LIN {X 0,Y 420.716,Z 380.039,A -85,B 0,C 180,E1 -10196.541,E2 -10196.541} C_VEL
LIN {X 0,Y 418.309,Z 369.381,A -85,B 0,C 180,E1 -10198.981,E2 -10198.981} C_VEL
LIN {X 0,Y 418.248,Z 369.386,A -85,B 0,C 180,E1 -10202.527,E2 -10202.527} C_VEL
LIN {X 0,Y 418.258,Z 369.383,A -85,B 0,C 180,E1 -10204.84,E2 -10204.84} C_VEL
LIN {X 0,Y 418.265,Z 369.379,A -85,B 0,C 180,E1 -10208.439,E2 -10208.439} C_VEL
LIN {X 0,Y 418.262,Z 369.382,A -85,B 0,C 180,E1 -10210.942,E2 -10210.942} C_VEL
LIN {X 0,Y 418.206,Z 369.391,A -85,B 0,C 180,E1 -10213.729,E2 -10213.729} C_VEL
LIN {X 0,Y 418.279,Z 369.382,A -85,B 0,C 180,E1 -10216.458,E2 -10216.458} C_VEL
LIN {X 0,Y 418.262,Z 369.383,A -85,B 0,C 180,E1 -10219.122,E2 -10219.122} C_VEL
LIN {X 0,Y 418.233,Z 369.387,A -85,B 0,C 180,E1 -10222.164,E2 -10222.164} C_VEL
LIN {X 0,Y 418.26,Z 369.385,A -85,B 0,C 180,E1 -10225.419,E2 -10225.419} C_VEL
LIN {X 0,Y 418.21,Z 369.387,A -85,B 0,C 180,E1 -10228.604,E2 -10228.604} C_VEL
LIN {X 0,Y 418.288,Z 369.381,A -85,B 0,C 180,E1 -10231.937,E2 -10231.937} C_VEL
LIN {X 0,Y 418.282,Z 369.378,A -85,B 0,C 180,E1 -10235.162,E2 -10235.162} C_VEL
LIN {X 0,Y 418.226,Z 369.382,A -85,B 0,C 180,E1 -10238.303,E2 -10238.303} C_VEL
LIN {X 0,Y 418.276,Z 369.385,A -85,B 0,C 180,E1 -10241.383,E2 -10241.383} C_VEL
LIN {X 0,Y 418.303,Z 369.376,A -85,B 0,C 180,E1 -10244.406,E2 -10244.406} C_VEL
LIN {X 0,Y 418.347,Z 369.369,A -85,B 0,C 180,E1 -10247.385,E2 -10247.385} C_VEL
LIN {X 0,Y 418.334,Z 369.373,A -85,B 0,C 180,E1 -10250.329,E2 -10250.329} C_VEL
LIN {X 0,Y 418.484,Z 369.351,A -85,B 0,C 180,E1 -10253.249,E2 -10253.249} C_VEL
LIN {X 0,Y 418.334,Z 369.377,A -85,B 0,C 180,E1 -10255.182,E2 -10255.182} C_VEL
LIN {X 0,Y 418.536,Z 369.344,A -85,B 0,C 180,E1 -10258.076,E2 -10258.076} C_VEL
LIN {X 0,Y 418.665,Z 369.332,A -85,B 0,C 180,E1 -10260,E2 -10260} C_VEL
LIN {X 0,Y 418.504,Z 369.347,A -85,B 0,C 180,E1 -10262.888,E2 -10262.888} C_VEL
LIN {X 0,Y 418.486,Z 369.354,A -85,B 0,C 180,E1 -10266.751,E2 -10266.751} C_VEL
LIN {X 0,Y 418.334,Z 369.375,A -85,B 0,C 180,E1 -10269.672,E2 -10269.672} C_VEL
LIN {X 0,Y 418.339,Z 369.371,A -85,B 0,C 180,E1 -10273.002,E2 -10273.002} C_VEL
LIN {X 0,Y 418.305,Z 369.373,A -85,B 0,C 180,E1 -10276.736,E2 -10276.736} C_VEL
LIN {X 0,Y 418.296,Z 369.374,A -85,B 0,C 180,E1 -10279.803,E2 -10279.803} C_VEL
LIN {X 0,Y 418.236,Z 369.389,A -85,B 0,C 180,E1 -10282.737,E2 -10282.737} C_VEL
LIN {X 0,Y 418.265,Z 369.382,A -85,B 0,C 180,E1 -10285.905,E2 -10285.905} C_VEL
LIN {X 0,Y 418.259,Z 369.385,A -85,B 0,C 180,E1 -10289.163,E2 -10289.163} C_VEL
LIN {X 0,Y 418.253,Z 369.384,A -85,B 0,C 180,E1 -10292.845,E2 -10292.845} C_VEL
LIN {X 0,Y 418.245,Z 369.385,A -85,B 0,C 180,E1 -10296.24,E2 -10296.24} C_VEL
LIN {X 0,Y 418.262,Z 369.381,A -85,B 0,C 180,E1 -10299.681,E2 -10299.681} C_VEL
LIN {X 0,Y 418.283,Z 369.377,A -85,B 0,C 180,E1 -10302.331,E2 -10302.331} C_VEL
LIN {X 0,Y 418.253,Z 369.383,A -85,B 0,C 180,E1 -10305.112,E2 -10305.112} C_VEL
LIN {X 0,Y 418.241,Z 369.385,A -85,B 0,C 180,E1 -10307.768,E2 -10307.768} C_VEL
LIN {X 0,Y 418.309,Z 369.47,A -85,B 0,C 180,E1 -10311.605,E2 -10311.605} C_VEL
LIN {X 0,Y 420.342,Z 380.03,A -85,B 0,C 180,E1 -10314.486,E2 -10314.486} C_VEL
LIN {X 0,Y 420.452,Z 381.221,A -85,B 0,C 180,E1 -10314.727,E2 -10314.727} C_VEL
LIN {X 0,Y 424.73,Z 398.892,A -85,B 0,C 180,E1 -10315.282,E2 -10315.282} C_VEL
LIN {X 0,Y 423.561,Z 487.472,A -85,B 0,C 180,E1 -10316.837,E2 -10316.837} C_VEL
LIN {X 0,Y 423.153,Z 500.671,A -85,B 0,C 180,E1 -10317.261,E2 -10317.261} C_VEL
LIN {X 0,Y 422.674,Z 513.047,A -85,B 0,C 180,E1 -10317.855,E2 -10317.855} C_VEL
LIN {X 0,Y 422.08,Z 523.932,A -85,B 0,C 180,E1 -10318.551,E2 -10318.551} C_VEL
LIN {X 0,Y 421.366,Z 534.615,A -85,B 0,C 180,E1 -10319.423,E2 -10319.423} C_VEL
LIN {X 0,Y 420.629,Z 544.481,A -85,B 0,C 180,E1 -10320.424,E2 -10320.424} C_VEL
LIN {X 0,Y 419.909,Z 553.272,A -85,B 0,C 180,E1 -10321.511,E2 -10321.511} C_VEL
LIN {X 0,Y 419.255,Z 561.69,A -85,B 0,C 180,E1 -10322.78,E2 -10322.78} C_VEL
LIN {X 0,Y 418.625,Z 568.972,A -85,B 0,C 180,E1 -10324.12,E2 -10324.12} C_VEL
LIN {X 0,Y 418.115,Z 575.775,A -85,B 0,C 180,E1 -10325.682,E2 -10325.682} C_VEL
LIN {X 0,Y 417.7,Z 581.039,A -85,B 0,C 180,E1 -10327.234,E2 -10327.234} C_VEL
LIN {X 0,Y 417.393,Z 585.027,A -85,B 0,C 180,E1 -10328.777,E2 -10328.777} C_VEL
LIN {X 0,Y 417.135,Z 588.367,A -85,B 0,C 180,E1 -10330.65,E2 -10330.65} C_VEL
LIN {X 0,Y 416.988,Z 590.049,A -85,B 0,C 180,E1 -10332.34,E2 -10332.34} C_VEL
LIN {X 0,Y 416.977,Z 590.52,A -85,B 0,C 180,E1 -10333.889,E2 -10333.889} C_VEL
LIN {X 0,Y 416.966,Z 590.033,A -85,B 0,C 180,E1 -10335.356,E2 -10335.356} C_VEL
LIN {X 0,Y 417.019,Z 589.173,A -85,B 0,C 180,E1 -10336.353,E2 -10336.353} C_VEL
LIN {X 0,Y 417.154,Z 587.301,A -85,B 0,C 180,E1 -10337.732,E2 -10337.732} C_VEL
LIN {X 0,Y 417.354,Z 584.039,A -85,B 0,C 180,E1 -10339.325,E2 -10339.325} C_VEL
LIN {X 0,Y 417.548,Z 579.915,A -85,B 0,C 180,E1 -10340.799,E2 -10340.799} C_VEL
LIN {X 0,Y 417.895,Z 574.601,A -85,B 0,C 180,E1 -10342.268,E2 -10342.268} C_VEL
LIN {X 0,Y 418.033,Z 572.633,A -85,B 0,C 180,E1 -10342.74,E2 -10342.74} C_VEL
LIN {X 0,Y 417.574,Z 569.57,A -85,B 0,C 180,E1 -10343.426,E2 -10343.426} C_VEL
LIN {X 0,Y 415.078,Z 564.217,A -85,B 0,C 180,E1 -10344.53,E2 -10344.53} C_VEL
LIN {X 0,Y 412.642,Z 558.354,A -85,B 0,C 180,E1 -10345.586,E2 -10345.586} C_VEL
LIN {X 0,Y 412.275,Z 554.353,A -85,B 0,C 180,E1 -10346.187,E2 -10346.187} C_VEL
LIN {X 0,Y 412.984,Z 544.392,A -85,B 0,C 180,E1 -10347.44,E2 -10347.44} C_VEL
LIN {X 0,Y 413.712,Z 533.485,A -85,B 0,C 180,E1 -10348.54,E2 -10348.54} C_VEL
LIN {X 0,Y 414.406,Z 522.256,A -85,B 0,C 180,E1 -10349.429,E2 -10349.429} C_VEL
LIN {X 0,Y 415,Z 509.859,A -85,B 0,C 180,E1 -10350.186,E2 -10350.186} C_VEL
LIN {X 0,Y 415.435,Z 497.781,A -85,B 0,C 180,E1 -10350.725,E2 -10350.725} C_VEL
LIN {X 0,Y 415.687,Z 484.799,A -85,B 0,C 180,E1 -10351.1,E2 -10351.1} C_VEL
LIN {X 0,Y 416.747,Z 399.82,A -85,B 0,C 180,E1 -10352.579,E2 -10352.579} C_VEL
LIN {X 0,Y 412.903,Z 380.764,A -85,B 0,C 180,E1 -10353.079,E2 -10353.079} C_VEL
LIN {X 0,Y 412.963,Z 379.392,A -85,B 0,C 180,E1 -10353.415,E2 -10353.415} C_VEL
LIN {X 0,Y 411.478,Z 370.232,A -85,B 0,C 180,E1 -10355.82,E2 -10355.82} C_VEL
LIN {X 0,Y 411.324,Z 370.25,A -85,B 0,C 180,E1 -10358.846,E2 -10358.846} C_VEL
LIN {X 0,Y 411.29,Z 370.251,A -85,B 0,C 180,E1 -10361.832,E2 -10361.832} C_VEL
LIN {X 0,Y 411.266,Z 370.254,A -85,B 0,C 180,E1 -10364.852,E2 -10364.852} C_VEL
LIN {X 0,Y 411.257,Z 370.254,A -85,B 0,C 180,E1 -10367.914,E2 -10367.914} C_VEL
LIN {X 0,Y 411.2,Z 370.264,A -85,B 0,C 180,E1 -10371.033,E2 -10371.033} C_VEL
LIN {X 0,Y 411.23,Z 370.256,A -85,B 0,C 180,E1 -10374.215,E2 -10374.215} C_VEL
LIN {X 0,Y 411.261,Z 370.257,A -85,B 0,C 180,E1 -10377.477,E2 -10377.477} C_VEL
LIN {X 0,Y 411.2,Z 370.263,A -85,B 0,C 180,E1 -10380.846,E2 -10380.846} C_VEL
LIN {X 0,Y 411.207,Z 370.259,A -85,B 0,C 180,E1 -10384.332,E2 -10384.332} C_VEL
LIN {X 0,Y 411.202,Z 370.26,A -85,B 0,C 180,E1 -10387.972,E2 -10387.972} C_VEL
LIN {X 0,Y 411.183,Z 370.263,A -85,B 0,C 180,E1 -10390.503,E2 -10390.503} C_VEL
LIN {X 0,Y 411.172,Z 370.27,A -85,B 0,C 180,E1 -10393.133,E2 -10393.133} C_VEL
LIN {X 0,Y 411.171,Z 370.264,A -85,B 0,C 180,E1 -10395.879,E2 -10395.879} C_VEL
LIN {X 0,Y 411.163,Z 370.269,A -85,B 0,C 180,E1 -10398.77,E2 -10398.77} C_VEL
LIN {X 0,Y 411.208,Z 370.259,A -85,B 0,C 180,E1 -10401.829,E2 -10401.829} C_VEL
LIN {X 0,Y 411.207,Z 370.264,A -85,B 0,C 180,E1 -10405.12,E2 -10405.12} C_VEL
LIN {X 0,Y 411.161,Z 370.265,A -85,B 0,C 180,E1 -10408.002,E2 -10408.002} C_VEL
LIN {X 0,Y 411.212,Z 370.26,A -85,B 0,C 180,E1 -10411.409,E2 -10411.409} C_VEL
LIN {X 0,Y 411.232,Z 370.256,A -85,B 0,C 180,E1 -10413.618,E2 -10413.618} C_VEL
LIN {X 0,Y 411.197,Z 370.267,A -85,B 0,C 180,E1 -10416.852,E2 -10416.852} C_VEL
LIN {X 0,Y 411.208,Z 370.26,A -85,B 0,C 180,E1 -10420.05,E2 -10420.05} C_VEL
LIN {X 0,Y 411.256,Z 370.256,A -85,B 0,C 180,E1 -10423.13,E2 -10423.13} C_VEL
LIN {X 0,Y 411.298,Z 370.252,A -85,B 0,C 180,E1 -10426.895,E2 -10426.895} C_VEL
LIN {X 0,Y 411.286,Z 370.251,A -85,B 0,C 180,E1 -10430.161,E2 -10430.161} C_VEL
LIN {X 0,Y 411.448,Z 370.231,A -85,B 0,C 180,E1 -10433.133,E2 -10433.133} C_VEL
LIN {X 0,Y 411.306,Z 370.249,A -85,B 0,C 180,E1 -10435.099,E2 -10435.099} C_VEL
LIN {X 0,Y 411.506,Z 370.224,A -85,B 0,C 180,E1 -10438.042,E2 -10438.042} C_VEL
LIN {X 0,Y 411.633,Z 370.208,A -85,B 0,C 180,E1 -10440,E2 -10440} C_VEL
LIN {X 0,Y 411.458,Z 370.23,A -85,B 0,C 180,E1 -10442.937,E2 -10442.937} C_VEL
LIN {X 0,Y 411.447,Z 370.232,A -85,B 0,C 180,E1 -10446.867,E2 -10446.867} C_VEL
LIN {X 0,Y 411.285,Z 370.251,A -85,B 0,C 180,E1 -10449.839,E2 -10449.839} C_VEL
LIN {X 0,Y 411.297,Z 370.248,A -85,B 0,C 180,E1 -10453.104,E2 -10453.104} C_VEL
LIN {X 0,Y 411.256,Z 370.255,A -85,B 0,C 180,E1 -10456.87,E2 -10456.87} C_VEL
LIN {X 0,Y 411.222,Z 370.261,A -85,B 0,C 180,E1 -10459.987,E2 -10459.987} C_VEL
LIN {X 0,Y 411.195,Z 370.261,A -85,B 0,C 180,E1 -10463.148,E2 -10463.148} C_VEL
LIN {X 0,Y 411.231,Z 370.262,A -85,B 0,C 180,E1 -10466.381,E2 -10466.381} C_VEL
LIN {X 0,Y 411.204,Z 370.262,A -85,B 0,C 180,E1 -10469.712,E2 -10469.712} C_VEL
LIN {X 0,Y 411.2,Z 370.26,A -85,B 0,C 180,E1 -10473.156,E2 -10473.156} C_VEL
LIN {X 0,Y 411.19,Z 370.264,A -85,B 0,C 180,E1 -10476.554,E2 -10476.554} C_VEL
LIN {X 0,Y 411.224,Z 370.26,A -85,B 0,C 180,E1 -10479.731,E2 -10479.731} C_VEL
LIN {X 0,Y 411.226,Z 370.257,A -85,B 0,C 180,E1 -10483.127,E2 -10483.127} C_VEL
LIN {X 0,Y 411.168,Z 370.27,A -85,B 0,C 180,E1 -10485.881,E2 -10485.881} C_VEL
LIN {X 0,Y 411.209,Z 370.261,A -85,B 0,C 180,E1 -10489.5,E2 -10489.5} C_VEL
LIN {X 0,Y 411.203,Z 370.266,A -85,B 0,C 180,E1 -10492.028,E2 -10492.028} C_VEL
LIN {X 0,Y 411.205,Z 370.264,A -85,B 0,C 180,E1 -10495.667,E2 -10495.667} C_VEL
LIN {X 0,Y 411.199,Z 370.261,A -85,B 0,C 180,E1 -10499.154,E2 -10499.154} C_VEL
LIN {X 0,Y 411.326,Z 370.37,A -85,B 0,C 180,E1 -10501.767,E2 -10501.767} C_VEL
LIN {X 0,Y 413.906,Z 383.596,A -85,B 0,C 180,E1 -10504.566,E2 -10504.566} C_VEL
LIN {X 0,Y 414.291,Z 387.926,A -85,B 0,C 180,E1 -10505.443,E2 -10505.443} C_VEL
LIN {X 0,Y 413.242,Z 404.064,A -85,B 0,C 180,E1 -10508.553,E2 -10508.553} C_VEL
LIN {X 0,Y 412.459,Z 416.368,A -85,B 0,C 180,E1 -10510.901,E2 -10510.901} C_VEL
LIN {X 0,Y 416.383,Z 444.904,A -85,B 0,C 180,E1 -10511.566,E2 -10511.566} C_VEL
LIN {X 0,Y 415.489,Z 524.864,A -85,B 0,C 180,E1 -10512.972,E2 -10512.972} C_VEL
LIN {X 0,Y 414.979,Z 538.176,A -85,B 0,C 180,E1 -10513.394,E2 -10513.394} C_VEL
LIN {X 0,Y 414.344,Z 550.959,A -85,B 0,C 180,E1 -10514.001,E2 -10514.001} C_VEL
LIN {X 0,Y 413.64,Z 562.314,A -85,B 0,C 180,E1 -10514.731,E2 -10514.731} C_VEL
LIN {X 0,Y 412.865,Z 574.043,A -85,B 0,C 180,E1 -10515.711,E2 -10515.711} C_VEL
LIN {X 0,Y 412.266,Z 583.918,A -85,B 0,C 180,E1 -10516.741,E2 -10516.741} C_VEL
LIN {X 0,Y 411.637,Z 593.223,A -85,B 0,C 180,E1 -10517.928,E2 -10517.928} C_VEL
LIN {X 0,Y 411.014,Z 601.161,A -85,B 0,C 180,E1 -10519.159,E2 -10519.159} C_VEL
LIN {X 0,Y 410.569,Z 608.912,A -85,B 0,C 180,E1 -10520.641,E2 -10520.641} C_VEL
LIN {X 0,Y 410.27,Z 615.134,A -85,B 0,C 180,E1 -10522.124,E2 -10522.124} C_VEL
LIN {X 0,Y 410.089,Z 620.393,A -85,B 0,C 180,E1 -10523.716,E2 -10523.716} C_VEL
LIN {X 0,Y 410.048,Z 623.859,A -85,B 0,C 180,E1 -10525.084,E2 -10525.084} C_VEL
LIN {X 0,Y 409.947,Z 625.807,A -85,B 0,C 180,E1 -10526.068,E2 -10526.068} C_VEL
LIN {X 0,Y 409.989,Z 627.336,A -85,B 0,C 180,E1 -10527.052,E2 -10527.052} C_VEL
LIN {X 0,Y 410.019,Z 628.405,A -85,B 0,C 180,E1 -10528.035,E2 -10528.035} C_VEL
LIN {X 0,Y 409.972,Z 629.35,A -85,B 0,C 180,E1 -10530,E2 -10530} C_VEL
LIN {X 0,Y 409.978,Z 629.236,A -85,B 0,C 180,E1 -10530.982,E2 -10530.982} C_VEL
LIN {X 0,Y 410.018,Z 628.688,A -85,B 0,C 180,E1 -10531.965,E2 -10531.965} C_VEL
LIN {X 0,Y 409.97,Z 627.738,A -85,B 0,C 180,E1 -10532.948,E2 -10532.948} C_VEL
LIN {X 0,Y 410.025,Z 624.641,A -85,B 0,C 180,E1 -10534.916,E2 -10534.916} C_VEL
LIN {X 0,Y 410.041,Z 621.58,A -85,B 0,C 180,E1 -10536.224,E2 -10536.224} C_VEL
LIN {X 0,Y 410.284,Z 616.556,A -85,B 0,C 180,E1 -10537.876,E2 -10537.876} C_VEL
LIN {X 0,Y 410.674,Z 609.634,A -85,B 0,C 180,E1 -10539.605,E2 -10539.605} C_VEL
LIN {X 0,Y 411.257,Z 602.158,A -85,B 0,C 180,E1 -10541.084,E2 -10541.084} C_VEL
LIN {X 0,Y 411.897,Z 594.555,A -85,B 0,C 180,E1 -10542.314,E2 -10542.314} C_VEL
LIN {X 0,Y 412.576,Z 585.369,A -85,B 0,C 180,E1 -10543.546,E2 -10543.546} C_VEL
LIN {X 0,Y 413.385,Z 575.315,A -85,B 0,C 180,E1 -10544.636,E2 -10544.636} C_VEL
LIN {X 0,Y 414.315,Z 563.918,A -85,B 0,C 180,E1 -10545.621,E2 -10545.621} C_VEL
LIN {X 0,Y 415.242,Z 551.273,A -85,B 0,C 180,E1 -10546.468,E2 -10546.468} C_VEL
LIN {X 0,Y 416.025,Z 538.172,A -85,B 0,C 180,E1 -10547.1,E2 -10547.1} C_VEL
LIN {X 0,Y 416.546,Z 525.252,A -85,B 0,C 180,E1 -10547.521,E2 -10547.521} C_VEL
LIN {X 0,Y 417.586,Z 444.003,A -85,B 0,C 180,E1 -10548.979,E2 -10548.979} C_VEL
LIN {X 0,Y 414.204,Z 422.378,A -85,B 0,C 180,E1 -10549.561,E2 -10549.561} C_VEL
LIN {X 0,Y 413.002,Z 415.847,A -85,B 0,C 180,E1 -10549.753,E2 -10549.753} C_VEL
LIN {X 0,Y 414.378,Z 397.592,A -85,B 0,C 180,E1 -10553.344,E2 -10553.344} C_VEL
LIN {X 0,Y 415.039,Z 389.085,A -85,B 0,C 180,E1 -10555.045,E2 -10555.045} C_VEL
LIN {X 0,Y 413.784,Z 381.321,A -85,B 0,C 180,E1 -10556.749,E2 -10556.749} C_VEL
LIN {X 0,Y 411.229,Z 370.261,A -85,B 0,C 180,E1 -10559.354,E2 -10559.354} C_VEL
LIN {X 0,Y 411.205,Z 370.26,A -85,B 0,C 180,E1 -10563.155,E2 -10563.155} C_VEL
LIN {X 0,Y 411.194,Z 370.267,A -85,B 0,C 180,E1 -10566.553,E2 -10566.553} C_VEL
LIN {X 0,Y 411.226,Z 370.26,A -85,B 0,C 180,E1 -10569.73,E2 -10569.73} C_VEL
LIN {X 0,Y 411.173,Z 370.263,A -85,B 0,C 180,E1 -10573.132,E2 -10573.132} C_VEL
LIN {X 0,Y 411.231,Z 370.261,A -85,B 0,C 180,E1 -10575.871,E2 -10575.871} C_VEL
LIN {X 0,Y 411.205,Z 370.262,A -85,B 0,C 180,E1 -10578.764,E2 -10578.764} C_VEL
LIN {X 0,Y 411.2,Z 370.264,A -85,B 0,C 180,E1 -10582.027,E2 -10582.027} C_VEL
LIN {X 0,Y 411.2,Z 370.264,A -85,B 0,C 180,E1 -10585.666,E2 -10585.666} C_VEL
LIN {X 0,Y 411.191,Z 370.263,A -85,B 0,C 180,E1 -10589.153,E2 -10589.153} C_VEL
LIN {X 0,Y 411.253,Z 370.254,A -85,B 0,C 180,E1 -10592.522,E2 -10592.522} C_VEL
LIN {X 0,Y 411.22,Z 370.264,A -85,B 0,C 180,E1 -10595.784,E2 -10595.784} C_VEL
LIN {X 0,Y 411.188,Z 370.258,A -85,B 0,C 180,E1 -10598.966,E2 -10598.966} C_VEL
LIN {X 0,Y 411.245,Z 370.251,A -85,B 0,C 180,E1 -10602.085,E2 -10602.085} C_VEL
LIN {X 0,Y 411.257,Z 370.257,A -85,B 0,C 180,E1 -10605.147,E2 -10605.147} C_VEL
LIN {X 0,Y 411.276,Z 370.249,A -85,B 0,C 180,E1 -10608.167,E2 -10608.167} C_VEL
LIN {X 0,Y 411.432,Z 370.225,A -85,B 0,C 180,E1 -10612.189,E2 -10612.189} C_VEL
LIN {X 0,Y 411.467,Z 370.228,A -85,B 0,C 180,E1 -10614.118,E2 -10614.118} C_VEL
LIN {X 0,Y 411.505,Z 370.22,A -85,B 0,C 180,E1 -10618.043,E2 -10618.043} C_VEL
LIN {X 0,Y 411.635,Z 370.208,A -85,B 0,C 180,E1 -10620,E2 -10620} C_VEL
LIN {X 0,Y 411.46,Z 370.224,A -85,B 0,C 180,E1 -10622.937,E2 -10622.937} C_VEL
LIN {X 0,Y 411.453,Z 370.23,A -85,B 0,C 180,E1 -10626.867,E2 -10626.867} C_VEL
LIN {X 0,Y 411.286,Z 370.251,A -85,B 0,C 180,E1 -10629.839,E2 -10629.839} C_VEL
LIN {X 0,Y 411.298,Z 370.249,A -85,B 0,C 180,E1 -10633.105,E2 -10633.105} C_VEL
LIN {X 0,Y 411.256,Z 370.252,A -85,B 0,C 180,E1 -10636.87,E2 -10636.87} C_VEL
LIN {X 0,Y 411.249,Z 370.251,A -85,B 0,C 180,E1 -10639.986,E2 -10639.986} C_VEL
LIN {X 0,Y 411.2,Z 370.262,A -85,B 0,C 180,E1 -10643.148,E2 -10643.148} C_VEL
LIN {X 0,Y 411.232,Z 370.259,A -85,B 0,C 180,E1 -10646.382,E2 -10646.382} C_VEL
LIN {X 0,Y 411.195,Z 370.261,A -85,B 0,C 180,E1 -10649.714,E2 -10649.714} C_VEL
LIN {X 0,Y 411.202,Z 370.257,A -85,B 0,C 180,E1 -10653.157,E2 -10653.157} C_VEL
LIN {X 0,Y 411.192,Z 370.266,A -85,B 0,C 180,E1 -10656.554,E2 -10656.554} C_VEL
LIN {X 0,Y 411.224,Z 370.258,A -85,B 0,C 180,E1 -10659.731,E2 -10659.731} C_VEL
LIN {X 0,Y 411.226,Z 370.262,A -85,B 0,C 180,E1 -10663.127,E2 -10663.127} C_VEL
LIN {X 0,Y 411.175,Z 370.266,A -85,B 0,C 180,E1 -10665.881,E2 -10665.881} C_VEL
LIN {X 0,Y 411.165,Z 370.271,A -85,B 0,C 180,E1 -10668.772,E2 -10668.772} C_VEL
LIN {X 0,Y 411.245,Z 370.355,A -85,B 0,C 180,E1 -10671.29,E2 -10671.29} C_VEL
LIN {X 0,Y 413.427,Z 381.383,A -85,B 0,C 180,E1 -10674.329,E2 -10674.329} C_VEL
LIN {X 0,Y 417.054,Z 395.122,A -85,B 0,C 180,E1 -10674.791,E2 -10674.791} C_VEL
LIN {X 0,Y 418.228,Z 400.694,A -85,B 0,C 180,E1 -10674.959,E2 -10674.959} C_VEL
LIN {X 0,Y 416.923,Z 487.236,A -85,B 0,C 180,E1 -10676.492,E2 -10676.492} C_VEL
LIN {X 0,Y 416.51,Z 500.636,A -85,B 0,C 180,E1 -10676.925,E2 -10676.925} C_VEL
LIN {X 0,Y 416.017,Z 512.437,A -85,B 0,C 180,E1 -10677.49,E2 -10677.49} C_VEL
LIN {X 0,Y 415.335,Z 524.449,A -85,B 0,C 180,E1 -10678.263,E2 -10678.263} C_VEL
LIN {X 0,Y 414.577,Z 535.101,A -85,B 0,C 180,E1 -10679.15,E2 -10679.15} C_VEL
LIN {X 0,Y 413.682,Z 546.359,A -85,B 0,C 180,E1 -10680.332,E2 -10680.332} C_VEL
LIN {X 0,Y 412.87,Z 555.591,A -85,B 0,C 180,E1 -10681.536,E2 -10681.536} C_VEL
LIN {X 0,Y 412.182,Z 563.863,A -85,B 0,C 180,E1 -10682.865,E2 -10682.865} C_VEL
LIN {X 0,Y 411.431,Z 571.792,A -85,B 0,C 180,E1 -10684.45,E2 -10684.45} C_VEL
LIN {X 0,Y 411.009,Z 577.104,A -85,B 0,C 180,E1 -10685.772,E2 -10685.772} C_VEL
LIN {X 0,Y 410.615,Z 581.904,A -85,B 0,C 180,E1 -10687.261,E2 -10687.261} C_VEL
LIN {X 0,Y 410.296,Z 585.943,A -85,B 0,C 180,E1 -10688.918,E2 -10688.918} C_VEL
LIN {X 0,Y 410.064,Z 588.629,A -85,B 0,C 180,E1 -10690.5,E2 -10690.5} C_VEL
LIN {X 0,Y 409.914,Z 590.203,A -85,B 0,C 180,E1 -10692.025,E2 -10692.025} C_VEL
LIN {X 0,Y 409.894,Z 590.853,A -85,B 0,C 180,E1 -10693.777,E2 -10693.777} C_VEL
LIN {X 0,Y 409.891,Z 590.487,A -85,B 0,C 180,E1 -10695.097,E2 -10695.097} C_VEL
LIN {X 0,Y 409.904,Z 589.756,A -85,B 0,C 180,E1 -10696.112,E2 -10696.112} C_VEL
LIN {X 0,Y 410.066,Z 587.775,A -85,B 0,C 180,E1 -10697.665,E2 -10697.665} C_VEL
LIN {X 0,Y 410.243,Z 584.921,A -85,B 0,C 180,E1 -10699.138,E2 -10699.138} C_VEL
LIN {X 0,Y 410.451,Z 580.973,A -85,B 0,C 180,E1 -10700.639,E2 -10700.639} C_VEL
LIN {X 0,Y 410.801,Z 575.871,A -85,B 0,C 180,E1 -10702.134,E2 -10702.134} C_VEL
LIN {X 0,Y 411.193,Z 569.457,A -85,B 0,C 180,E1 -10703.622,E2 -10703.622} C_VEL
LIN {X 0,Y 411.758,Z 561.444,A -85,B 0,C 180,E1 -10705.104,E2 -10705.104} C_VEL
LIN {X 0,Y 412.275,Z 554.353,A -85,B 0,C 180,E1 -10706.187,E2 -10706.187} C_VEL
LIN {X 0,Y 411.937,Z 550.209,A -85,B 0,C 180,E1 -10706.764,E2 -10706.764} C_VEL
LIN {X 0,Y 409.649,Z 543.204,A -85,B 0,C 180,E1 -10707.689,E2 -10707.689} C_VEL
LIN {X 0,Y 407.351,Z 535.723,A -85,B 0,C 180,E1 -10708.546,E2 -10708.546} C_VEL
LIN {X 0,Y 406.998,Z 530.789,A -85,B 0,C 180,E1 -10709.011,E2 -10709.011} C_VEL
LIN {X 0,Y 407.728,Z 519.319,A -85,B 0,C 180,E1 -10709.878,E2 -10709.878} C_VEL
LIN {X 0,Y 408.226,Z 506.943,A -85,B 0,C 180,E1 -10710.585,E2 -10710.585} C_VEL
LIN {X 0,Y 408.664,Z 493.988,A -85,B 0,C 180,E1 -10711.109,E2 -10711.109} C_VEL
LIN {X 0,Y 408.949,Z 481.779,A -85,B 0,C 180,E1 -10711.416,E2 -10711.416} C_VEL
LIN {X 0,Y 409.897,Z 400.575,A -85,B 0,C 180,E1 -10712.845,E2 -10712.845} C_VEL
LIN {X 0,Y 405.956,Z 381.024,A -85,B 0,C 180,E1 -10713.377,E2 -10713.377} C_VEL
LIN {X 0,Y 404.398,Z 371.113,A -85,B 0,C 180,E1 -10715.985,E2 -10715.985} C_VEL
LIN {X 0,Y 404.271,Z 371.129,A -85,B 0,C 180,E1 -10719.001,E2 -10719.001} C_VEL
LIN {X 0,Y 404.262,Z 371.125,A -85,B 0,C 180,E1 -10722.041,E2 -10722.041} C_VEL
LIN {X 0,Y 404.212,Z 371.135,A -85,B 0,C 180,E1 -10725.117,E2 -10725.117} C_VEL
LIN {X 0,Y 404.214,Z 371.13,A -85,B 0,C 180,E1 -10728.237,E2 -10728.237} C_VEL
LIN {X 0,Y 404.164,Z 371.142,A -85,B 0,C 180,E1 -10731.417,E2 -10731.417} C_VEL
LIN {X 0,Y 404.18,Z 371.136,A -85,B 0,C 180,E1 -10734.665,E2 -10734.665} C_VEL
LIN {X 0,Y 404.198,Z 371.133,A -85,B 0,C 180,E1 -10737.999,E2 -10737.999} C_VEL
LIN {X 0,Y 404.148,Z 371.141,A -85,B 0,C 180,E1 -10741.559,E2 -10741.559} C_VEL
LIN {X 0,Y 404.186,Z 371.139,A -85,B 0,C 180,E1 -10745.015,E2 -10745.015} C_VEL
LIN {X 0,Y 404.16,Z 371.14,A -85,B 0,C 180,E1 -10748.755,E2 -10748.755} C_VEL
LIN {X 0,Y 404.122,Z 371.143,A -85,B 0,C 180,E1 -10751.599,E2 -10751.599} C_VEL
LIN {X 0,Y 404.145,Z 371.141,A -85,B 0,C 180,E1 -10754.521,E2 -10754.521} C_VEL
LIN {X 0,Y 404.137,Z 371.143,A -85,B 0,C 180,E1 -10757.295,E2 -10757.295} C_VEL
LIN {X 0,Y 404.166,Z 371.136,A -85,B 0,C 180,E1 -10759.954,E2 -10759.954} C_VEL
LIN {X 0,Y 404.137,Z 371.145,A -85,B 0,C 180,E1 -10763.123,E2 -10763.123} C_VEL
LIN {X 0,Y 404.141,Z 371.14,A -85,B 0,C 180,E1 -10766.187,E2 -10766.187} C_VEL
LIN {X 0,Y 404.14,Z 371.14,A -85,B 0,C 180,E1 -10769.714,E2 -10769.714} C_VEL
LIN {X 0,Y 404.19,Z 371.137,A -85,B 0,C 180,E1 -10773.122,E2 -10773.122} C_VEL
LIN {X 0,Y 404.171,Z 371.137,A -85,B 0,C 180,E1 -10775.334,E2 -10775.334} C_VEL
LIN {X 0,Y 404.132,Z 371.145,A -85,B 0,C 180,E1 -10778.58,E2 -10778.58} C_VEL
LIN {X 0,Y 404.203,Z 371.132,A -85,B 0,C 180,E1 -10781.761,E2 -10781.761} C_VEL
LIN {X 0,Y 404.201,Z 371.137,A -85,B 0,C 180,E1 -10784.881,E2 -10784.881} C_VEL
LIN {X 0,Y 404.25,Z 371.126,A -85,B 0,C 180,E1 -10787.958,E2 -10787.958} C_VEL
LIN {X 0,Y 404.397,Z 371.109,A -85,B 0,C 180,E1 -10792.128,E2 -10792.128} C_VEL
LIN {X 0,Y 404.416,Z 371.106,A -85,B 0,C 180,E1 -10794.015,E2 -10794.015} C_VEL
LIN {X 0,Y 404.475,Z 371.099,A -85,B 0,C 180,E1 -10798.008,E2 -10798.008} C_VEL
LIN {X 0,Y 404.602,Z 371.084,A -85,B 0,C 180,E1 -10800,E2 -10800} C_VEL
LIN {X 0,Y 404.415,Z 371.107,A -85,B 0,C 180,E1 -10802.988,E2 -10802.988} C_VEL
LIN {X 0,Y 404.394,Z 371.109,A -85,B 0,C 180,E1 -10806.987,E2 -10806.987} C_VEL
LIN {X 0,Y 404.251,Z 371.128,A -85,B 0,C 180,E1 -10810.012,E2 -10810.012} C_VEL
LIN {X 0,Y 404.258,Z 371.125,A -85,B 0,C 180,E1 -10813.211,E2 -10813.211} C_VEL
LIN {X 0,Y 404.211,Z 371.131,A -85,B 0,C 180,E1 -10817.009,E2 -10817.009} C_VEL
LIN {X 0,Y 404.156,Z 371.144,A -85,B 0,C 180,E1 -10820.352,E2 -10820.352} C_VEL
LIN {X 0,Y 404.162,Z 371.137,A -85,B 0,C 180,E1 -10823.575,E2 -10823.575} C_VEL
LIN {X 0,Y 404.176,Z 371.137,A -85,B 0,C 180,E1 -10825.767,E2 -10825.767} C_VEL
LIN {X 0,Y 404.191,Z 371.138,A -85,B 0,C 180,E1 -10828,E2 -10828} C_VEL
LIN {X 0,Y 404.136,Z 371.141,A -85,B 0,C 180,E1 -10831.559,E2 -10831.559} C_VEL
LIN {X 0,Y 404.179,Z 371.135,A -85,B 0,C 180,E1 -10835.017,E2 -10835.017} C_VEL
LIN {X 0,Y 404.159,Z 371.138,A -85,B 0,C 180,E1 -10838.756,E2 -10838.756} C_VEL
LIN {X 0,Y 404.187,Z 371.136,A -85,B 0,C 180,E1 -10841.611,E2 -10841.611} C_VEL
LIN {X 0,Y 404.188,Z 371.135,A -85,B 0,C 180,E1 -10844.53,E2 -10844.53} C_VEL
LIN {X 0,Y 404.167,Z 371.137,A -85,B 0,C 180,E1 -10847.301,E2 -10847.301} C_VEL
LIN {X 0,Y 404.166,Z 371.143,A -85,B 0,C 180,E1 -10849.956,E2 -10849.956} C_VEL
LIN {X 0,Y 404.139,Z 371.14,A -85,B 0,C 180,E1 -10853.125,E2 -10853.125} C_VEL
LIN {X 0,Y 404.144,Z 371.143,A -85,B 0,C 180,E1 -10856.189,E2 -10856.189} C_VEL
LIN {X 0,Y 404.154,Z 371.143,A -85,B 0,C 180,E1 -10859.716,E2 -10859.716} C_VEL
LIN {X 0,Y 404.288,Z 371.281,A -85,B 0,C 180,E1 -10861.549,E2 -10861.549} C_VEL
LIN {X 0,Y 407.143,Z 385.98,A -85,B 0,C 180,E1 -10864.709,E2 -10864.709} C_VEL
LIN {X 0,Y 407.255,Z 390.057,A -85,B 0,C 180,E1 -10865.534,E2 -10865.534} C_VEL
LIN {X 0,Y 406.01,Z 408.698,A -85,B 0,C 180,E1 -10869.186,E2 -10869.186} C_VEL
LIN {X 0,Y 405.489,Z 415.994,A -85,B 0,C 180,E1 -10870.601,E2 -10870.601} C_VEL
LIN {X 0,Y 409.529,Z 445.893,A -85,B 0,C 180,E1 -10871.316,E2 -10871.316} C_VEL
LIN {X 0,Y 408.602,Z 525.289,A -85,B 0,C 180,E1 -10872.741,E2 -10872.741} C_VEL
LIN {X 0,Y 408.032,Z 539.122,A -85,B 0,C 180,E1 -10873.2,E2 -10873.2} C_VEL
LIN {X 0,Y 407.383,Z 552.054,A -85,B 0,C 180,E1 -10873.849,E2 -10873.849} C_VEL
LIN {X 0,Y 406.533,Z 564.644,A -85,B 0,C 180,E1 -10874.714,E2 -10874.714} C_VEL
LIN {X 0,Y 405.781,Z 575.888,A -85,B 0,C 180,E1 -10875.712,E2 -10875.712} C_VEL
LIN {X 0,Y 405.159,Z 585.405,A -85,B 0,C 180,E1 -10876.764,E2 -10876.764} C_VEL
LIN {X 0,Y 404.526,Z 594.315,A -85,B 0,C 180,E1 -10877.967,E2 -10877.967} C_VEL
LIN {X 0,Y 403.79,Z 603.361,A -85,B 0,C 180,E1 -10879.47,E2 -10879.47} C_VEL
LIN {X 0,Y 403.38,Z 610.652,A -85,B 0,C 180,E1 -10880.979,E2 -10880.979} C_VEL
LIN {X 0,Y 403.129,Z 616.466,A -85,B 0,C 180,E1 -10882.487,E2 -10882.487} C_VEL
LIN {X 0,Y 402.966,Z 621.033,A -85,B 0,C 180,E1 -10883.993,E2 -10883.993} C_VEL
LIN {X 0,Y 402.956,Z 623.439,A -85,B 0,C 180,E1 -10884.997,E2 -10884.997} C_VEL
LIN {X 0,Y 402.868,Z 625.401,A -85,B 0,C 180,E1 -10885.999,E2 -10885.999} C_VEL
LIN {X 0,Y 402.889,Z 626.948,A -85,B 0,C 180,E1 -10887,E2 -10887} C_VEL
LIN {X 0,Y 402.948,Z 628.04,A -85,B 0,C 180,E1 -10888.001,E2 -10888.001} C_VEL
LIN {X 0,Y 402.894,Z 629.01,A -85,B 0,C 180,E1 -10890,E2 -10890} C_VEL
LIN {X 0,Y 402.903,Z 628.912,A -85,B 0,C 180,E1 -10890.999,E2 -10890.999} C_VEL
LIN {X 0,Y 402.946,Z 628.385,A -85,B 0,C 180,E1 -10891.999,E2 -10891.999} C_VEL
LIN {X 0,Y 402.861,Z 626.115,A -85,B 0,C 180,E1 -10894.001,E2 -10894.001} C_VEL
LIN {X 0,Y 402.92,Z 623.31,A -85,B 0,C 180,E1 -10895.505,E2 -10895.505} C_VEL
LIN {X 0,Y 403.076,Z 619.486,A -85,B 0,C 180,E1 -10897.01,E2 -10897.01} C_VEL
LIN {X 0,Y 403.327,Z 614.546,A -85,B 0,C 180,E1 -10898.517,E2 -10898.517} C_VEL
LIN {X 0,Y 403.74,Z 608.346,A -85,B 0,C 180,E1 -10900.024,E2 -10900.024} C_VEL
LIN {X 0,Y 404.371,Z 600.664,A -85,B 0,C 180,E1 -10901.529,E2 -10901.529} C_VEL
LIN {X 0,Y 405.253,Z 591.044,A -85,B 0,C 180,E1 -10903.029,E2 -10903.029} C_VEL
LIN {X 0,Y 406.019,Z 581.601,A -85,B 0,C 180,E1 -10904.225,E2 -10904.225} C_VEL
LIN {X 0,Y 406.88,Z 571.444,A -85,B 0,C 180,E1 -10905.272,E2 -10905.272} C_VEL
LIN {X 0,Y 407.743,Z 560.981,A -85,B 0,C 180,E1 -10906.137,E2 -10906.137} C_VEL
LIN {X 0,Y 408.714,Z 548.417,A -85,B 0,C 180,E1 -10906.932,E2 -10906.932} C_VEL
LIN {X 0,Y 409.439,Z 535.188,A -85,B 0,C 180,E1 -10907.545,E2 -10907.545} C_VEL
LIN {X 0,Y 409.938,Z 523.093,A -85,B 0,C 180,E1 -10907.909,E2 -10907.909} C_VEL
LIN {X 0,Y 410.998,Z 445.092,A -85,B 0,C 180,E1 -10909.318,E2 -10909.318} C_VEL
LIN {X 0,Y 407.997,Z 425.446,A -85,B 0,C 180,E1 -10909.856,E2 -10909.856} C_VEL
LIN {X 0,Y 406.159,Z 415.386,A -85,B 0,C 180,E1 -10910.174,E2 -10910.174} C_VEL
LIN {X 0,Y 407.625,Z 397.233,A -85,B 0,C 180,E1 -10913.821,E2 -10913.821} C_VEL
LIN {X 0,Y 408.159,Z 390.365,A -85,B 0,C 180,E1 -10915.224,E2 -10915.224} C_VEL
LIN {X 0,Y 406.856,Z 382.607,A -85,B 0,C 180,E1 -10916.964,E2 -10916.964} C_VEL
LIN {X 0,Y 404.177,Z 371.139,A -85,B 0,C 180,E1 -10919.705,E2 -10919.705} C_VEL
LIN {X 0,Y 404.169,Z 371.136,A -85,B 0,C 180,E1 -10923.419,E2 -10923.419} C_VEL
LIN {X 0,Y 404.142,Z 371.145,A -85,B 0,C 180,E1 -10926.245,E2 -10926.245} C_VEL
LIN {X 0,Y 404.162,Z 371.136,A -85,B 0,C 180,E1 -10928.755,E2 -10928.755} C_VEL
LIN {X 0,Y 404.146,Z 371.138,A -85,B 0,C 180,E1 -10931.603,E2 -10931.603} C_VEL
LIN {X 0,Y 404.149,Z 371.141,A -85,B 0,C 180,E1 -10934.523,E2 -10934.523} C_VEL
LIN {X 0,Y 404.206,Z 371.135,A -85,B 0,C 180,E1 -10937.305,E2 -10937.305} C_VEL
LIN {X 0,Y 404.164,Z 371.14,A -85,B 0,C 180,E1 -10939.955,E2 -10939.955} C_VEL
LIN {X 0,Y 404.135,Z 371.14,A -85,B 0,C 180,E1 -10943.124,E2 -10943.124} C_VEL
LIN {X 0,Y 404.139,Z 371.139,A -85,B 0,C 180,E1 -10946.187,E2 -10946.187} C_VEL
LIN {X 0,Y 404.147,Z 371.139,A -85,B 0,C 180,E1 -10949.715,E2 -10949.715} C_VEL
LIN {X 0,Y 404.188,Z 371.135,A -85,B 0,C 180,E1 -10953.122,E2 -10953.122} C_VEL
LIN {X 0,Y 404.17,Z 371.137,A -85,B 0,C 180,E1 -10955.334,E2 -10955.334} C_VEL
LIN {X 0,Y 404.13,Z 371.136,A -85,B 0,C 180,E1 -10958.58,E2 -10958.58} C_VEL
LIN {X 0,Y 404.202,Z 371.132,A -85,B 0,C 180,E1 -10961.762,E2 -10961.762} C_VEL
LIN {X 0,Y 404.203,Z 371.133,A -85,B 0,C 180,E1 -10964.882,E2 -10964.882} C_VEL
LIN {X 0,Y 404.248,Z 371.125,A -85,B 0,C 180,E1 -10967.958,E2 -10967.958} C_VEL
LIN {X 0,Y 404.397,Z 371.101,A -85,B 0,C 180,E1 -10972.129,E2 -10972.129} C_VEL
LIN {X 0,Y 404.415,Z 371.107,A -85,B 0,C 180,E1 -10974.015,E2 -10974.015} C_VEL
LIN {X 0,Y 404.474,Z 371.096,A -85,B 0,C 180,E1 -10978.009,E2 -10978.009} C_VEL
LIN {X 0,Y 404.605,Z 371.084,A -85,B 0,C 180,E1 -10980,E2 -10980} C_VEL
LIN {X 0,Y 404.417,Z 371.101,A -85,B 0,C 180,E1 -10982.989,E2 -10982.989} C_VEL
LIN {X 0,Y 404.399,Z 371.107,A -85,B 0,C 180,E1 -10986.988,E2 -10986.988} C_VEL
LIN {X 0,Y 404.252,Z 371.127,A -85,B 0,C 180,E1 -10990.012,E2 -10990.012} C_VEL
LIN {X 0,Y 404.259,Z 371.128,A -85,B 0,C 180,E1 -10993.212,E2 -10993.212} C_VEL
LIN {X 0,Y 404.209,Z 371.131,A -85,B 0,C 180,E1 -10997.008,E2 -10997.008} C_VEL
LIN {X 0,Y 404.199,Z 371.13,A -85,B 0,C 180,E1 -11000.35,E2 -11000.35} C_VEL
LIN {X 0,Y 404.165,Z 371.134,A -85,B 0,C 180,E1 -11003.575,E2 -11003.575} C_VEL
LIN {X 0,Y 404.19,Z 371.137,A -85,B 0,C 180,E1 -11006.878,E2 -11006.878} C_VEL
LIN {X 0,Y 404.14,Z 371.141,A -85,B 0,C 180,E1 -11010.286,E2 -11010.286} C_VEL
LIN {X 0,Y 404.141,Z 371.133,A -85,B 0,C 180,E1 -11013.813,E2 -11013.813} C_VEL
LIN {X 0,Y 404.137,Z 371.147,A -85,B 0,C 180,E1 -11016.877,E2 -11016.877} C_VEL
LIN {X 0,Y 404.164,Z 371.138,A -85,B 0,C 180,E1 -11020.084,E2 -11020.084} C_VEL
LIN {X 0,Y 404.2,Z 371.136,A -85,B 0,C 180,E1 -11023.092,E2 -11023.092} C_VEL
LIN {X 0,Y 404.154,Z 371.141,A -85,B 0,C 180,E1 -11025.928,E2 -11025.928} C_VEL
LIN {X 0,Y 404.12,Z 371.149,A -85,B 0,C 180,E1 -11028.636,E2 -11028.636} C_VEL
LIN {X 0,Y 404.214,Z 371.285,A -85,B 0,C 180,E1 -11030.971,E2 -11030.971} C_VEL
LIN {X 0,Y 406.279,Z 381.621,A -85,B 0,C 180,E1 -11033.895,E2 -11033.895} C_VEL
LIN {X 0,Y 408.917,Z 389.695,A -85,B 0,C 180,E1 -11034.219,E2 -11034.219} C_VEL
LIN {X 0,Y 411.627,Z 401.542,A -85,B 0,C 180,E1 -11034.601,E2 -11034.601} C_VEL
LIN {X 0,Y 410.282,Z 488.315,A -85,B 0,C 180,E1 -11036.172,E2 -11036.172} C_VEL
LIN {X 0,Y 409.817,Z 501.426,A -85,B 0,C 180,E1 -11036.608,E2 -11036.608} C_VEL
LIN {X 0,Y 409.305,Z 513.346,A -85,B 0,C 180,E1 -11037.196,E2 -11037.196} C_VEL
LIN {X 0,Y 408.623,Z 524.486,A -85,B 0,C 180,E1 -11037.926,E2 -11037.926} C_VEL
LIN {X 0,Y 407.809,Z 535.636,A -85,B 0,C 180,E1 -11038.869,E2 -11038.869} C_VEL
LIN {X 0,Y 406.858,Z 546.954,A -85,B 0,C 180,E1 -11040.081,E2 -11040.081} C_VEL
LIN {X 0,Y 406.008,Z 556.061,A -85,B 0,C 180,E1 -11041.292,E2 -11041.292} C_VEL
LIN {X 0,Y 405.253,Z 564.29,A -85,B 0,C 180,E1 -11042.641,E2 -11042.641} C_VEL
LIN {X 0,Y 404.483,Z 572.199,A -85,B 0,C 180,E1 -11044.255,E2 -11044.255} C_VEL
LIN {X 0,Y 403.913,Z 578.442,A -85,B 0,C 180,E1 -11045.865,E2 -11045.865} C_VEL
LIN {X 0,Y 403.52,Z 583.262,A -85,B 0,C 180,E1 -11047.471,E2 -11047.471} C_VEL
LIN {X 0,Y 403.212,Z 586.833,A -85,B 0,C 180,E1 -11049.065,E2 -11049.065} C_VEL
LIN {X 0,Y 402.974,Z 589.296,A -85,B 0,C 180,E1 -11050.649,E2 -11050.649} C_VEL
LIN {X 0,Y 402.844,Z 590.344,A -85,B 0,C 180,E1 -11051.698,E2 -11051.698} C_VEL
LIN {X 0,Y 402.812,Z 591.179,A -85,B 0,C 180,E1 -11053.661,E2 -11053.661} C_VEL
LIN {X 0,Y 402.802,Z 590.942,A -85,B 0,C 180,E1 -11054.828,E2 -11054.828} C_VEL
LIN {X 0,Y 402.817,Z 590.288,A -85,B 0,C 180,E1 -11055.862,E2 -11055.862} C_VEL
LIN {X 0,Y 402.967,Z 588.231,A -85,B 0,C 180,E1 -11057.604,E2 -11057.604} C_VEL
LIN {X 0,Y 403.197,Z 584.644,A -85,B 0,C 180,E1 -11059.454,E2 -11059.454} C_VEL
LIN {X 0,Y 403.439,Z 580.497,A -85,B 0,C 180,E1 -11060.98,E2 -11060.98} C_VEL
LIN {X 0,Y 403.861,Z 574.302,A -85,B 0,C 180,E1 -11062.715,E2 -11062.715} C_VEL
LIN {X 0,Y 404.357,Z 567.253,A -85,B 0,C 180,E1 -11064.264,E2 -11064.264} C_VEL
LIN {X 0,Y 405.002,Z 558.615,A -85,B 0,C 180,E1 -11065.771,E2 -11065.771} C_VEL
LIN {X 0,Y 405.625,Z 549.767,A -85,B 0,C 180,E1 -11067.021,E2 -11067.021} C_VEL
LIN {X 0,Y 406.409,Z 540.012,A -85,B 0,C 180,E1 -11068.142,E2 -11068.142} C_VEL
LIN {X 0,Y 406.998,Z 530.789,A -85,B 0,C 180,E1 -11069.011,E2 -11069.011} C_VEL
LIN {X 0,Y 406.63,Z 525.753,A -85,B 0,C 180,E1 -11069.447,E2 -11069.447} C_VEL
LIN {X 0,Y 404.273,Z 517.436,A -85,B 0,C 180,E1 -11070.142,E2 -11070.142} C_VEL
LIN {X 0,Y 401.901,Z 508.786,A -85,B 0,C 180,E1 -11070.74,E2 -11070.74} C_VEL
LIN {X 0,Y 401.494,Z 503.237,A -85,B 0,C 180,E1 -11071.018,E2 -11071.018} C_VEL
LIN {X 0,Y 401.892,Z 489.499,A -85,B 0,C 180,E1 -11071.503,E2 -11071.503} C_VEL
LIN {X 0,Y 402.388,Z 458.74,A -85,B 0,C 180,E1 -11072.089,E2 -11072.089} C_VEL
LIN {X 0,Y 403.061,Z 401.428,A -85,B 0,C 180,E1 -11073.118,E2 -11073.118} C_VEL
LIN {X 0,Y 398.874,Z 381.375,A -85,B 0,C 180,E1 -11073.671,E2 -11073.671} C_VEL
LIN {X 0,Y 397.338,Z 371.993,A -85,B 0,C 180,E1 -11076.219,E2 -11076.219} C_VEL
LIN {X 0,Y 397.241,Z 372.005,A -85,B 0,C 180,E1 -11079.162,E2 -11079.162} C_VEL
LIN {X 0,Y 397.225,Z 372.001,A -85,B 0,C 180,E1 -11082.258,E2 -11082.258} C_VEL
LIN {X 0,Y 397.184,Z 372.013,A -85,B 0,C 180,E1 -11085.391,E2 -11085.391} C_VEL
LIN {X 0,Y 397.166,Z 372.009,A -85,B 0,C 180,E1 -11088.573,E2 -11088.573} C_VEL
LIN {X 0,Y 397.113,Z 372.017,A -85,B 0,C 180,E1 -11091.817,E2 -11091.817} C_VEL
LIN {X 0,Y 397.156,Z 372.013,A -85,B 0,C 180,E1 -11095.512,E2 -11095.512} C_VEL
LIN {X 0,Y 397.126,Z 372.014,A -85,B 0,C 180,E1 -11098.543,E2 -11098.543} C_VEL
LIN {X 0,Y 397.084,Z 372.018,A -85,B 0,C 180,E1 -11102.07,E2 -11102.07} C_VEL
LIN {X 0,Y 397.121,Z 372.017,A -85,B 0,C 180,E1 -11105.503,E2 -11105.503} C_VEL
LIN {X 0,Y 397.134,Z 372.017,A -85,B 0,C 180,E1 -11108.861,E2 -11108.861} C_VEL
LIN {X 0,Y 397.067,Z 372.021,A -85,B 0,C 180,E1 -11112.266,E2 -11112.266} C_VEL
LIN {X 0,Y 397.089,Z 372.025,A -85,B 0,C 180,E1 -11115.067,E2 -11115.067} C_VEL
LIN {X 0,Y 397.066,Z 372.021,A -85,B 0,C 180,E1 -11118.02,E2 -11118.02} C_VEL
LIN {X 0,Y 397.131,Z 372.018,A -85,B 0,C 180,E1 -11121.137,E2 -11121.137} C_VEL
LIN {X 0,Y 397.116,Z 372.017,A -85,B 0,C 180,E1 -11124.496,E2 -11124.496} C_VEL
LIN {X 0,Y 397.073,Z 372.02,A -85,B 0,C 180,E1 -11127.927,E2 -11127.927} C_VEL
LIN {X 0,Y 397.116,Z 372.016,A -85,B 0,C 180,E1 -11131.455,E2 -11131.455} C_VEL
LIN {X 0,Y 397.147,Z 372.014,A -85,B 0,C 180,E1 -11134.487,E2 -11134.487} C_VEL
LIN {X 0,Y 397.103,Z 372.02,A -85,B 0,C 180,E1 -11137.085,E2 -11137.085} C_VEL
LIN {X 0,Y 397.141,Z 372.014,A -85,B 0,C 180,E1 -11140.352,E2 -11140.352} C_VEL
LIN {X 0,Y 397.159,Z 372.009,A -85,B 0,C 180,E1 -11143.552,E2 -11143.552} C_VEL
LIN {X 0,Y 397.221,Z 372.008,A -85,B 0,C 180,E1 -11146.702,E2 -11146.702} C_VEL
LIN {X 0,Y 397.211,Z 372.003,A -85,B 0,C 180,E1 -11149.808,E2 -11149.808} C_VEL
LIN {X 0,Y 397.345,Z 371.99,A -85,B 0,C 180,E1 -11152.888,E2 -11152.888} C_VEL
LIN {X 0,Y 397.249,Z 372.001,A -85,B 0,C 180,E1 -11154.925,E2 -11154.925} C_VEL
LIN {X 0,Y 397.443,Z 371.975,A -85,B 0,C 180,E1 -11157.973,E2 -11157.973} C_VEL
LIN {X 0,Y 397.572,Z 371.959,A -85,B 0,C 180,E1 -11160,E2 -11160} C_VEL
LIN {X 0,Y 397.374,Z 371.984,A -85,B 0,C 180,E1 -11163.041,E2 -11163.041} C_VEL
LIN {X 0,Y 397.365,Z 371.986,A -85,B 0,C 180,E1 -11166.091,E2 -11166.091} C_VEL
LIN {X 0,Y 397.245,Z 371.999,A -85,B 0,C 180,E1 -11169.162,E2 -11169.162} C_VEL
LIN {X 0,Y 397.211,Z 372.008,A -85,B 0,C 180,E1 -11172.258,E2 -11172.258} C_VEL
LIN {X 0,Y 397.175,Z 372.007,A -85,B 0,C 180,E1 -11175.392,E2 -11175.392} C_VEL
LIN {X 0,Y 397.154,Z 372.014,A -85,B 0,C 180,E1 -11178.574,E2 -11178.574} C_VEL
LIN {X 0,Y 397.089,Z 372.02,A -85,B 0,C 180,E1 -11181.819,E2 -11181.819} C_VEL
LIN {X 0,Y 397.149,Z 372.01,A -85,B 0,C 180,E1 -11185.132,E2 -11185.132} C_VEL
LIN {X 0,Y 397.157,Z 372.012,A -85,B 0,C 180,E1 -11187.777,E2 -11187.777} C_VEL
LIN {X 0,Y 397.077,Z 372.02,A -85,B 0,C 180,E1 -11190.882,E2 -11190.882} C_VEL
LIN {X 0,Y 397.12,Z 372.017,A -85,B 0,C 180,E1 -11194.494,E2 -11194.494} C_VEL
LIN {X 0,Y 397.105,Z 372.021,A -85,B 0,C 180,E1 -11198.275,E2 -11198.275} C_VEL
LIN {X 0,Y 397.152,Z 372.016,A -85,B 0,C 180,E1 -11201.994,E2 -11201.994} C_VEL
LIN {X 0,Y 397.108,Z 372.016,A -85,B 0,C 180,E1 -11205.066,E2 -11205.066} C_VEL
LIN {X 0,Y 397.106,Z 372.023,A -85,B 0,C 180,E1 -11208.015,E2 -11208.015} C_VEL
LIN {X 0,Y 397.136,Z 372.012,A -85,B 0,C 180,E1 -11211.138,E2 -11211.138} C_VEL
LIN {X 0,Y 397.118,Z 372.016,A -85,B 0,C 180,E1 -11214.497,E2 -11214.497} C_VEL
LIN {X 0,Y 397.11,Z 372.022,A -85,B 0,C 180,E1 -11217.932,E2 -11217.932} C_VEL
LIN {X 0,Y 397.226,Z 372.178,A -85,B 0,C 180,E1 -11221.321,E2 -11221.321} C_VEL
LIN {X 0,Y 399.842,Z 385.344,A -85,B 0,C 180,E1 -11224.213,E2 -11224.213} C_VEL
LIN {X 0,Y 400.401,Z 389.459,A -85,B 0,C 180,E1 -11225.087,E2 -11225.087} C_VEL
LIN {X 0,Y 399.255,Z 405.59,A -85,B 0,C 180,E1 -11228.306,E2 -11228.306} C_VEL
LIN {X 0,Y 398.573,Z 415.95,A -85,B 0,C 180,E1 -11230.317,E2 -11230.317} C_VEL
LIN {X 0,Y 402.691,Z 446.385,A -85,B 0,C 180,E1 -11231.052,E2 -11231.052} C_VEL
LIN {X 0,Y 401.749,Z 524.322,A -85,B 0,C 180,E1 -11232.47,E2 -11232.47} C_VEL
LIN {X 0,Y 401.239,Z 537.607,A -85,B 0,C 180,E1 -11232.907,E2 -11232.907} C_VEL
LIN {X 0,Y 400.567,Z 549.803,A -85,B 0,C 180,E1 -11233.501,E2 -11233.501} C_VEL
LIN {X 0,Y 399.775,Z 562.116,A -85,B 0,C 180,E1 -11234.319,E2 -11234.319} C_VEL
LIN {X 0,Y 398.899,Z 573.763,A -85,B 0,C 180,E1 -11235.33,E2 -11235.33} C_VEL
LIN {X 0,Y 398.288,Z 583.466,A -85,B 0,C 180,E1 -11236.383,E2 -11236.383} C_VEL
LIN {X 0,Y 397.531,Z 593.691,A -85,B 0,C 180,E1 -11237.752,E2 -11237.752} C_VEL
LIN {X 0,Y 396.78,Z 602.794,A -85,B 0,C 180,E1 -11239.282,E2 -11239.282} C_VEL
LIN {X 0,Y 396.336,Z 610.132,A -85,B 0,C 180,E1 -11240.817,E2 -11240.817} C_VEL
LIN {X 0,Y 396.056,Z 615.994,A -85,B 0,C 180,E1 -11242.352,E2 -11242.352} C_VEL
LIN {X 0,Y 395.855,Z 621.264,A -85,B 0,C 180,E1 -11244.156,E2 -11244.156} C_VEL
LIN {X 0,Y 395.79,Z 624.995,A -85,B 0,C 180,E1 -11245.927,E2 -11245.927} C_VEL
LIN {X 0,Y 395.791,Z 626.557,A -85,B 0,C 180,E1 -11246.946,E2 -11246.946} C_VEL
LIN {X 0,Y 395.878,Z 627.674,A -85,B 0,C 180,E1 -11247.965,E2 -11247.965} C_VEL
LIN {X 0,Y 395.819,Z 628.669,A -85,B 0,C 180,E1 -11250,E2 -11250} C_VEL
LIN {X 0,Y 395.83,Z 628.585,A -85,B 0,C 180,E1 -11251.017,E2 -11251.017} C_VEL
LIN {X 0,Y 395.856,Z 628.081,A -85,B 0,C 180,E1 -11252.035,E2 -11252.035} C_VEL
LIN {X 0,Y 395.783,Z 625.837,A -85,B 0,C 180,E1 -11254.073,E2 -11254.073} C_VEL
LIN {X 0,Y 395.828,Z 622.628,A -85,B 0,C 180,E1 -11255.808,E2 -11255.808} C_VEL
LIN {X 0,Y 396.063,Z 617.78,A -85,B 0,C 180,E1 -11257.648,E2 -11257.648} C_VEL
LIN {X 0,Y 396.455,Z 611.459,A -85,B 0,C 180,E1 -11259.438,E2 -11259.438} C_VEL
LIN {X 0,Y 396.983,Z 604.601,A -85,B 0,C 180,E1 -11260.971,E2 -11260.971} C_VEL
LIN {X 0,Y 397.866,Z 596.083,A -85,B 0,C 180,E1 -11262.497,E2 -11262.497} C_VEL
LIN {X 0,Y 398.672,Z 586.352,A -85,B 0,C 180,E1 -11263.9,E2 -11263.9} C_VEL
LIN {X 0,Y 399.649,Z 575.566,A -85,B 0,C 180,E1 -11265.151,E2 -11265.151} C_VEL
LIN {X 0,Y 400.684,Z 564.414,A -85,B 0,C 180,E1 -11266.167,E2 -11266.167} C_VEL
LIN {X 0,Y 401.694,Z 552.087,A -85,B 0,C 180,E1 -11267.041,E2 -11267.041} C_VEL
LIN {X 0,Y 402.51,Z 540.418,A -85,B 0,C 180,E1 -11267.66,E2 -11267.66} C_VEL
LIN {X 0,Y 403.147,Z 527.943,A -85,B 0,C 180,E1 -11268.123,E2 -11268.123} C_VEL
LIN {X 0,Y 403.499,Z 511.052,A -85,B 0,C 180,E1 -11268.491,E2 -11268.491} C_VEL
LIN {X 0,Y 404.418,Z 445.893,A -85,B 0,C 180,E1 -11269.676,E2 -11269.676} C_VEL
LIN {X 0,Y 401.49,Z 426.761,A -85,B 0,C 180,E1 -11270.216,E2 -11270.216} C_VEL
LIN {X 0,Y 399.296,Z 414.959,A -85,B 0,C 180,E1 -11270.61,E2 -11270.61} C_VEL
LIN {X 0,Y 400.796,Z 397.941,A -85,B 0,C 180,E1 -11274.096,E2 -11274.096} C_VEL
LIN {X 0,Y 401.28,Z 391.651,A -85,B 0,C 180,E1 -11275.409,E2 -11275.409} C_VEL
LIN {X 0,Y 399.408,Z 381.524,A -85,B 0,C 180,E1 -11277.755,E2 -11277.755} C_VEL
LIN {X 0,Y 397.12,Z 372.021,A -85,B 0,C 180,E1 -11280.119,E2 -11280.119} C_VEL
LIN {X 0,Y 397.117,Z 372.016,A -85,B 0,C 180,E1 -11283.717,E2 -11283.717} C_VEL
LIN {X 0,Y 397.097,Z 372.021,A -85,B 0,C 180,E1 -11287.209,E2 -11287.209} C_VEL
LIN {X 0,Y 397.119,Z 372.019,A -85,B 0,C 180,E1 -11290.448,E2 -11290.448} C_VEL
LIN {X 0,Y 397.1,Z 372.019,A -85,B 0,C 180,E1 -11293.647,E2 -11293.647} C_VEL
LIN {X 0,Y 397.16,Z 372.012,A -85,B 0,C 180,E1 -11296.511,E2 -11296.511} C_VEL
LIN {X 0,Y 397.119,Z 372.02,A -85,B 0,C 180,E1 -11299.55,E2 -11299.55} C_VEL
LIN {X 0,Y 397.094,Z 372.017,A -85,B 0,C 180,E1 -11302.789,E2 -11302.789} C_VEL
LIN {X 0,Y 397.112,Z 372.013,A -85,B 0,C 180,E1 -11306.282,E2 -11306.282} C_VEL
LIN {X 0,Y 397.107,Z 372.015,A -85,B 0,C 180,E1 -11310.133,E2 -11310.133} C_VEL
LIN {X 0,Y 397.188,Z 372.005,A -85,B 0,C 180,E1 -11312.609,E2 -11312.609} C_VEL
LIN {X 0,Y 397.125,Z 372.017,A -85,B 0,C 180,E1 -11315.981,E2 -11315.981} C_VEL
LIN {X 0,Y 397.131,Z 372.017,A -85,B 0,C 180,E1 -11319.704,E2 -11319.704} C_VEL
LIN {X 0,Y 397.176,Z 372.002,A -85,B 0,C 180,E1 -11322.844,E2 -11322.844} C_VEL
LIN {X 0,Y 397.171,Z 372.012,A -85,B 0,C 180,E1 -11325.657,E2 -11325.657} C_VEL
LIN {X 0,Y 397.191,Z 372.003,A -85,B 0,C 180,E1 -11328.777,E2 -11328.777} C_VEL
LIN {X 0,Y 397.353,Z 371.979,A -85,B 0,C 180,E1 -11332.075,E2 -11332.075} C_VEL
LIN {X 0,Y 397.248,Z 372.001,A -85,B 0,C 180,E1 -11334.925,E2 -11334.925} C_VEL
LIN {X 0,Y 397.443,Z 371.972,A -85,B 0,C 180,E1 -11337.973,E2 -11337.973} C_VEL
LIN {X 0,Y 397.574,Z 371.96,A -85,B 0,C 180,E1 -11340,E2 -11340} C_VEL
LIN {X 0,Y 397.376,Z 371.979,A -85,B 0,C 180,E1 -11343.042,E2 -11343.042} C_VEL
LIN {X 0,Y 397.342,Z 371.983,A -85,B 0,C 180,E1 -11346.655,E2 -11346.655} C_VEL
LIN {X 0,Y 397.246,Z 372.003,A -85,B 0,C 180,E1 -11349.162,E2 -11349.162} C_VEL
LIN {X 0,Y 397.212,Z 371.997,A -85,B 0,C 180,E1 -11352.259,E2 -11352.259} C_VEL
LIN {X 0,Y 397.173,Z 372.007,A -85,B 0,C 180,E1 -11355.393,E2 -11355.393} C_VEL
LIN {X 0,Y 397.165,Z 372.012,A -85,B 0,C 180,E1 -11358.574,E2 -11358.574} C_VEL
LIN {X 0,Y 397.121,Z 372.016,A -85,B 0,C 180,E1 -11361.818,E2 -11361.818} C_VEL
LIN {X 0,Y 397.147,Z 372.014,A -85,B 0,C 180,E1 -11365.513,E2 -11365.513} C_VEL
LIN {X 0,Y 397.117,Z 372.018,A -85,B 0,C 180,E1 -11368.545,E2 -11368.545} C_VEL
LIN {X 0,Y 397.073,Z 372.023,A -85,B 0,C 180,E1 -11372.073,E2 -11372.073} C_VEL
LIN {X 0,Y 397.116,Z 372.017,A -85,B 0,C 180,E1 -11375.505,E2 -11375.505} C_VEL
LIN {X 0,Y 397.134,Z 372.019,A -85,B 0,C 180,E1 -11378.864,E2 -11378.864} C_VEL
LIN {X 0,Y 397.157,Z 372.007,A -85,B 0,C 180,E1 -11382.256,E2 -11382.256} C_VEL
LIN {X 0,Y 397.112,Z 372.016,A -85,B 0,C 180,E1 -11385.066,E2 -11385.066} C_VEL
LIN {X 0,Y 397.067,Z 372.023,A -85,B 0,C 180,E1 -11388.022,E2 -11388.022} C_VEL
LIN {X 0,Y 397.177,Z 372.19,A -85,B 0,C 180,E1 -11390.622,E2 -11390.622} C_VEL
LIN {X 0,Y 399.142,Z 381.97,A -85,B 0,C 180,E1 -11393.457,E2 -11393.457} C_VEL
LIN {X 0,Y 402.169,Z 390.238,A -85,B 0,C 180,E1 -11393.816,E2 -11393.816} C_VEL
LIN {X 0,Y 405.077,Z 402.671,A -85,B 0,C 180,E1 -11394.234,E2 -11394.234} C_VEL
LIN {X 0,Y 403.658,Z 488.204,A -85,B 0,C 180,E1 -11395.804,E2 -11395.804} C_VEL
LIN {X 0,Y 403.179,Z 501.776,A -85,B 0,C 180,E1 -11396.261,E2 -11396.261} C_VEL
LIN {X 0,Y 402.669,Z 513.254,A -85,B 0,C 180,E1 -11396.835,E2 -11396.835} C_VEL
LIN {X 0,Y 401.889,Z 525.085,A -85,B 0,C 180,E1 -11397.62,E2 -11397.62} C_VEL
LIN {X 0,Y 401.031,Z 536.167,A -85,B 0,C 180,E1 -11398.577,E2 -11398.577} C_VEL
LIN {X 0,Y 400.027,Z 547.447,A -85,B 0,C 180,E1 -11399.808,E2 -11399.808} C_VEL
LIN {X 0,Y 399.156,Z 556.529,A -85,B 0,C 180,E1 -11401.041,E2 -11401.041} C_VEL
LIN {X 0,Y 398.325,Z 564.898,A -85,B 0,C 180,E1 -11402.444,E2 -11402.444} C_VEL
LIN {X 0,Y 397.479,Z 573.083,A -85,B 0,C 180,E1 -11404.16,E2 -11404.16} C_VEL
LIN {X 0,Y 396.834,Z 579.725,A -85,B 0,C 180,E1 -11405.963,E2 -11405.963} C_VEL
LIN {X 0,Y 396.414,Z 584.439,A -85,B 0,C 180,E1 -11407.654,E2 -11407.654} C_VEL
LIN {X 0,Y 396.103,Z 587.667,A -85,B 0,C 180,E1 -11409.216,E2 -11409.216} C_VEL
LIN {X 0,Y 395.94,Z 589.309,A -85,B 0,C 180,E1 -11410.291,E2 -11410.291} C_VEL
LIN {X 0,Y 395.798,Z 590.489,A -85,B 0,C 180,E1 -11411.361,E2 -11411.361} C_VEL
LIN {X 0,Y 395.738,Z 591.198,A -85,B 0,C 180,E1 -11412.428,E2 -11412.428} C_VEL
LIN {X 0,Y 395.731,Z 591.504,A -85,B 0,C 180,E1 -11413.542,E2 -11413.542} C_VEL
LIN {X 0,Y 395.727,Z 591.387,A -85,B 0,C 180,E1 -11414.55,E2 -11414.55} C_VEL
LIN {X 0,Y 395.729,Z 590.817,A -85,B 0,C 180,E1 -11415.604,E2 -11415.604} C_VEL
LIN {X 0,Y 395.87,Z 588.684,A -85,B 0,C 180,E1 -11417.539,E2 -11417.539} C_VEL
LIN {X 0,Y 396.096,Z 585.524,A -85,B 0,C 180,E1 -11419.263,E2 -11419.263} C_VEL
LIN {X 0,Y 396.32,Z 581.553,A -85,B 0,C 180,E1 -11420.817,E2 -11420.817} C_VEL
LIN {X 0,Y 396.72,Z 576.23,A -85,B 0,C 180,E1 -11422.416,E2 -11422.416} C_VEL
LIN {X 0,Y 397.12,Z 569.972,A -85,B 0,C 180,E1 -11423.905,E2 -11423.905} C_VEL
LIN {X 0,Y 397.776,Z 561.912,A -85,B 0,C 180,E1 -11425.44,E2 -11425.44} C_VEL
LIN {X 0,Y 398.422,Z 553.701,A -85,B 0,C 180,E1 -11426.714,E2 -11426.714} C_VEL
LIN {X 0,Y 399.203,Z 543.675,A -85,B 0,C 180,E1 -11427.982,E2 -11427.982} C_VEL
LIN {X 0,Y 399.879,Z 533.753,A -85,B 0,C 180,E1 -11428.993,E2 -11428.993} C_VEL
LIN {X 0,Y 400.601,Z 522.84,A -85,B 0,C 180,E1 -11429.882,E2 -11429.882} C_VEL
LIN {X 0,Y 401.202,Z 511.513,A -85,B 0,C 180,E1 -11430.603,E2 -11430.603} C_VEL
LIN {X 0,Y 401.494,Z 503.237,A -85,B 0,C 180,E1 -11431.018,E2 -11431.018} C_VEL
LIN {X 0,Y 401.005,Z 499.471,A -85,B 0,C 180,E1 -11431.199,E2 -11431.199} C_VEL
LIN {X 0,Y 398.389,Z 493.623,A -85,B 0,C 180,E1 -11431.517,E2 -11431.517} C_VEL
LIN {X 0,Y 395.756,Z 487.71,A -85,B 0,C 180,E1 -11431.797,E2 -11431.797} C_VEL
LIN {X 0,Y 395.194,Z 483.849,A -85,B 0,C 180,E1 -11431.906,E2 -11431.906} C_VEL
LIN {X 0,Y 396.199,Z 402.031,A -85,B 0,C 180,E1 -11433.4,E2 -11433.4} C_VEL
LIN {X 0,Y 392.525,Z 384.316,A -85,B 0,C 180,E1 -11433.897,E2 -11433.897} C_VEL
LIN {X 0,Y 391.719,Z 381.657,A -85,B 0,C 180,E1 -11433.999,E2 -11433.999} C_VEL
LIN {X 0,Y 390.299,Z 372.869,A -85,B 0,C 180,E1 -11436.397,E2 -11436.397} C_VEL
LIN {X 0,Y 390.198,Z 372.883,A -85,B 0,C 180,E1 -11439.329,E2 -11439.329} C_VEL
LIN {X 0,Y 390.176,Z 372.879,A -85,B 0,C 180,E1 -11442.483,E2 -11442.483} C_VEL
LIN {X 0,Y 390.144,Z 372.886,A -85,B 0,C 180,E1 -11445.676,E2 -11445.676} C_VEL
LIN {X 0,Y 390.11,Z 372.89,A -85,B 0,C 180,E1 -11448.921,E2 -11448.921} C_VEL
LIN {X 0,Y 390.051,Z 372.895,A -85,B 0,C 180,E1 -11452.233,E2 -11452.233} C_VEL
LIN {X 0,Y 390.122,Z 372.888,A -85,B 0,C 180,E1 -11455.743,E2 -11455.743} C_VEL
LIN {X 0,Y 390.065,Z 372.899,A -85,B 0,C 180,E1 -11459.108,E2 -11459.108} C_VEL
LIN {X 0,Y 390.046,Z 372.897,A -85,B 0,C 180,E1 -11462.72,E2 -11462.72} C_VEL
LIN {X 0,Y 390.058,Z 372.894,A -85,B 0,C 180,E1 -11465.825,E2 -11465.825} C_VEL
LIN {X 0,Y 390.072,Z 372.897,A -85,B 0,C 180,E1 -11469.218,E2 -11469.218} C_VEL
LIN {X 0,Y 390.041,Z 372.897,A -85,B 0,C 180,E1 -11472.373,E2 -11472.373} C_VEL
LIN {X 0,Y 390.045,Z 372.899,A -85,B 0,C 180,E1 -11475.354,E2 -11475.354} C_VEL
LIN {X 0,Y 390.03,Z 372.897,A -85,B 0,C 180,E1 -11478.186,E2 -11478.186} C_VEL
LIN {X 0,Y 390.09,Z 372.896,A -85,B 0,C 180,E1 -11480.907,E2 -11480.907} C_VEL
LIN {X 0,Y 390.082,Z 372.896,A -85,B 0,C 180,E1 -11484.792,E2 -11484.792} C_VEL
LIN {X 0,Y 390.019,Z 372.901,A -85,B 0,C 180,E1 -11488.495,E2 -11488.495} C_VEL
LIN {X 0,Y 390.112,Z 372.887,A -85,B 0,C 180,E1 -11492.069,E2 -11492.069} C_VEL
LIN {X 0,Y 390.074,Z 372.892,A -85,B 0,C 180,E1 -11495.518,E2 -11495.518} C_VEL
LIN {X 0,Y 390.049,Z 372.9,A -85,B 0,C 180,E1 -11498.877,E2 -11498.877} C_VEL
LIN {X 0,Y 390.121,Z 372.887,A -85,B 0,C 180,E1 -11502.166,E2 -11502.166} C_VEL
LIN {X 0,Y 390.14,Z 372.884,A -85,B 0,C 180,E1 -11505.392,E2 -11505.392} C_VEL
LIN {X 0,Y 390.142,Z 372.889,A -85,B 0,C 180,E1 -11508.571,E2 -11508.571} C_VEL
LIN {X 0,Y 390.3,Z 372.865,A -85,B 0,C 180,E1 -11512.031,E2 -11512.031} C_VEL
LIN {X 0,Y 390.221,Z 372.878,A -85,B 0,C 180,E1 -11514.833,E2 -11514.833} C_VEL
LIN {X 0,Y 390.412,Z 372.851,A -85,B 0,C 180,E1 -11517.936,E2 -11517.936} C_VEL
LIN {X 0,Y 390.541,Z 372.835,A -85,B 0,C 180,E1 -11520,E2 -11520} C_VEL
LIN {X 0,Y 390.308,Z 372.864,A -85,B 0,C 180,E1 -11523.096,E2 -11523.096} C_VEL
LIN {X 0,Y 390.319,Z 372.865,A -85,B 0,C 180,E1 -11526.202,E2 -11526.202} C_VEL
LIN {X 0,Y 390.197,Z 372.877,A -85,B 0,C 180,E1 -11529.329,E2 -11529.329} C_VEL
LIN {X 0,Y 390.186,Z 372.878,A -85,B 0,C 180,E1 -11533.439,E2 -11533.439} C_VEL
LIN {X 0,Y 390.142,Z 372.883,A -85,B 0,C 180,E1 -11537.309,E2 -11537.309} C_VEL
LIN {X 0,Y 390.079,Z 372.896,A -85,B 0,C 180,E1 -11540.47,E2 -11540.47} C_VEL
LIN {X 0,Y 390.082,Z 372.891,A -85,B 0,C 180,E1 -11543.351,E2 -11543.351} C_VEL
LIN {X 0,Y 390.106,Z 372.889,A -85,B 0,C 180,E1 -11546.769,E2 -11546.769} C_VEL
LIN {X 0,Y 390.037,Z 372.902,A -85,B 0,C 180,E1 -11550.3,E2 -11550.3} C_VEL
LIN {X 0,Y 390.062,Z 372.899,A -85,B 0,C 180,E1 -11554.025,E2 -11554.025} C_VEL
LIN {X 0,Y 390.042,Z 372.897,A -85,B 0,C 180,E1 -11557.552,E2 -11557.552} C_VEL
LIN {X 0,Y 390.078,Z 372.892,A -85,B 0,C 180,E1 -11560.827,E2 -11560.827} C_VEL
LIN {X 0,Y 390.101,Z 372.894,A -85,B 0,C 180,E1 -11563.895,E2 -11563.895} C_VEL
LIN {X 0,Y 390.077,Z 372.894,A -85,B 0,C 180,E1 -11567.62,E2 -11567.62} C_VEL
LIN {X 0,Y 390.093,Z 372.889,A -85,B 0,C 180,E1 -11570.909,E2 -11570.909} C_VEL
LIN {X 0,Y 390.084,Z 372.891,A -85,B 0,C 180,E1 -11574.794,E2 -11574.794} C_VEL
LIN {X 0,Y 390.046,Z 372.896,A -85,B 0,C 180,E1 -11578.499,E2 -11578.499} C_VEL
LIN {X 0,Y 390.163,Z 373.078,A -85,B 0,C 180,E1 -11581.085,E2 -11581.085} C_VEL
LIN {X 0,Y 392.569,Z 384.863,A -85,B 0,C 180,E1 -11583.734,E2 -11583.734} C_VEL
LIN {X 0,Y 393.406,Z 390.202,A -85,B 0,C 180,E1 -11584.896,E2 -11584.896} C_VEL
LIN {X 0,Y 392.624,Z 400.954,A -85,B 0,C 180,E1 -11587.088,E2 -11587.088} C_VEL
LIN {X 0,Y 391.601,Z 415.351,A -85,B 0,C 180,E1 -11589.995,E2 -11589.995} C_VEL
LIN {X 0,Y 395.861,Z 446.555,A -85,B 0,C 180,E1 -11590.775,E2 -11590.775} C_VEL
LIN {X 0,Y 394.867,Z 524.495,A -85,B 0,C 180,E1 -11592.221,E2 -11592.221} C_VEL
LIN {X 0,Y 394.31,Z 538.38,A -85,B 0,C 180,E1 -11592.697,E2 -11592.697} C_VEL
LIN {X 0,Y 393.59,Z 550.831,A -85,B 0,C 180,E1 -11593.333,E2 -11593.333} C_VEL
LIN {X 0,Y 392.781,Z 562.759,A -85,B 0,C 180,E1 -11594.165,E2 -11594.165} C_VEL
LIN {X 0,Y 391.881,Z 574.228,A -85,B 0,C 180,E1 -11595.194,E2 -11595.194} C_VEL
LIN {X 0,Y 391.207,Z 584.429,A -85,B 0,C 180,E1 -11596.342,E2 -11596.342} C_VEL
LIN {X 0,Y 390.522,Z 593.035,A -85,B 0,C 180,E1 -11597.529,E2 -11597.529} C_VEL
LIN {X 0,Y 389.766,Z 602.197,A -85,B 0,C 180,E1 -11599.087,E2 -11599.087} C_VEL
LIN {X 0,Y 389.289,Z 609.581,A -85,B 0,C 180,E1 -11600.649,E2 -11600.649} C_VEL
LIN {X 0,Y 388.984,Z 615.491,A -85,B 0,C 180,E1 -11602.212,E2 -11602.212} C_VEL
LIN {X 0,Y 388.834,Z 620.137,A -85,B 0,C 180,E1 -11603.774,E2 -11603.774} C_VEL
LIN {X 0,Y 388.781,Z 622.584,A -85,B 0,C 180,E1 -11604.814,E2 -11604.814} C_VEL
LIN {X 0,Y 388.715,Z 624.579,A -85,B 0,C 180,E1 -11605.853,E2 -11605.853} C_VEL
LIN {X 0,Y 388.695,Z 626.156,A -85,B 0,C 180,E1 -11606.891,E2 -11606.891} C_VEL
LIN {X 0,Y 388.79,Z 627.304,A -85,B 0,C 180,E1 -11607.928,E2 -11607.928} C_VEL
LIN {X 0,Y 388.76,Z 628.011,A -85,B 0,C 180,E1 -11608.964,E2 -11608.964} C_VEL
LIN {X 0,Y 388.746,Z 628.328,A -85,B 0,C 180,E1 -11610,E2 -11610} C_VEL
LIN {X 0,Y 388.759,Z 628.258,A -85,B 0,C 180,E1 -11611.036,E2 -11611.036} C_VEL
LIN {X 0,Y 388.754,Z 627.782,A -85,B 0,C 180,E1 -11612.072,E2 -11612.072} C_VEL
LIN {X 0,Y 388.708,Z 625.57,A -85,B 0,C 180,E1 -11614.147,E2 -11614.147} C_VEL
LIN {X 0,Y 388.744,Z 623.863,A -85,B 0,C 180,E1 -11615.186,E2 -11615.186} C_VEL
LIN {X 0,Y 388.842,Z 620.446,A -85,B 0,C 180,E1 -11616.747,E2 -11616.747} C_VEL
LIN {X 0,Y 389.112,Z 615.963,A -85,B 0,C 180,E1 -11618.308,E2 -11618.308} C_VEL
LIN {X 0,Y 389.602,Z 609.207,A -85,B 0,C 180,E1 -11620.13,E2 -11620.13} C_VEL
LIN {X 0,Y 390.277,Z 601.864,A -85,B 0,C 180,E1 -11621.688,E2 -11621.688} C_VEL
LIN {X 0,Y 391.24,Z 592.784,A -85,B 0,C 180,E1 -11623.24,E2 -11623.24} C_VEL
LIN {X 0,Y 392.059,Z 583.413,A -85,B 0,C 180,E1 -11624.534,E2 -11624.534} C_VEL
LIN {X 0,Y 393.091,Z 573.041,A -85,B 0,C 180,E1 -11625.689,E2 -11625.689} C_VEL
LIN {X 0,Y 394.181,Z 561.554,A -85,B 0,C 180,E1 -11626.708,E2 -11626.708} C_VEL
LIN {X 0,Y 395.215,Z 549.502,A -85,B 0,C 180,E1 -11627.529,E2 -11627.529} C_VEL
LIN {X 0,Y 396.059,Z 536.149,A -85,B 0,C 180,E1 -11628.191,E2 -11628.191} C_VEL
LIN {X 0,Y 396.656,Z 522.889,A -85,B 0,C 180,E1 -11628.626,E2 -11628.626} C_VEL
LIN {X 0,Y 397.854,Z 446.696,A -85,B 0,C 180,E1 -11630.051,E2 -11630.051} C_VEL
LIN {X 0,Y 394.791,Z 426.754,A -85,B 0,C 180,E1 -11630.629,E2 -11630.629} C_VEL
LIN {X 0,Y 392.487,Z 414.739,A -85,B 0,C 180,E1 -11631.022,E2 -11631.022} C_VEL
LIN {X 0,Y 394.188,Z 396.465,A -85,B 0,C 180,E1 -11634.846,E2 -11634.846} C_VEL
LIN {X 0,Y 394.386,Z 392.941,A -85,B 0,C 180,E1 -11635.603,E2 -11635.603} C_VEL
LIN {X 0,Y 392.439,Z 382.76,A -85,B 0,C 180,E1 -11638.019,E2 -11638.019} C_VEL
LIN {X 0,Y 390.081,Z 372.897,A -85,B 0,C 180,E1 -11640.52,E2 -11640.52} C_VEL
LIN {X 0,Y 390.066,Z 372.897,A -85,B 0,C 180,E1 -11644.024,E2 -11644.024} C_VEL
LIN {X 0,Y 390.045,Z 372.9,A -85,B 0,C 180,E1 -11647.551,E2 -11647.551} C_VEL
LIN {X 0,Y 390.075,Z 372.894,A -85,B 0,C 180,E1 -11650.824,E2 -11650.824} C_VEL
LIN {X 0,Y 390.056,Z 372.9,A -85,B 0,C 180,E1 -11653.886,E2 -11653.886} C_VEL
LIN {X 0,Y 390.113,Z 372.889,A -85,B 0,C 180,E1 -11656.797,E2 -11656.797} C_VEL
LIN {X 0,Y 390.073,Z 372.898,A -85,B 0,C 180,E1 -11659.563,E2 -11659.563} C_VEL
LIN {X 0,Y 390.042,Z 372.896,A -85,B 0,C 180,E1 -11662.448,E2 -11662.448} C_VEL
LIN {X 0,Y 390.062,Z 372.893,A -85,B 0,C 180,E1 -11666.045,E2 -11666.045} C_VEL
LIN {X 0,Y 390.045,Z 372.894,A -85,B 0,C 180,E1 -11669.867,E2 -11669.867} C_VEL
LIN {X 0,Y 390.107,Z 372.89,A -85,B 0,C 180,E1 -11673.231,E2 -11673.231} C_VEL
LIN {X 0,Y 390.099,Z 372.889,A -85,B 0,C 180,E1 -11676.75,E2 -11676.75} C_VEL
LIN {X 0,Y 390.096,Z 372.893,A -85,B 0,C 180,E1 -11679.983,E2 -11679.983} C_VEL
LIN {X 0,Y 390.133,Z 372.881,A -85,B 0,C 180,E1 -11683.248,E2 -11683.248} C_VEL
LIN {X 0,Y 390.186,Z 372.876,A -85,B 0,C 180,E1 -11686.561,E2 -11686.561} C_VEL
LIN {X 0,Y 390.197,Z 372.878,A -85,B 0,C 180,E1 -11690.671,E2 -11690.671} C_VEL
LIN {X 0,Y 390.319,Z 372.865,A -85,B 0,C 180,E1 -11693.798,E2 -11693.798} C_VEL
LIN {X 0,Y 390.412,Z 372.847,A -85,B 0,C 180,E1 -11697.937,E2 -11697.937} C_VEL
LIN {X 0,Y 390.543,Z 372.835,A -85,B 0,C 180,E1 -11700,E2 -11700} C_VEL
LIN {X 0,Y 390.31,Z 372.859,A -85,B 0,C 180,E1 -11703.097,E2 -11703.097} C_VEL
LIN {X 0,Y 390.296,Z 372.861,A -85,B 0,C 180,E1 -11706.651,E2 -11706.651} C_VEL
LIN {X 0,Y 390.198,Z 372.883,A -85,B 0,C 180,E1 -11709.329,E2 -11709.329} C_VEL
LIN {X 0,Y 390.187,Z 372.883,A -85,B 0,C 180,E1 -11713.439,E2 -11713.439} C_VEL
LIN {X 0,Y 390.142,Z 372.886,A -85,B 0,C 180,E1 -11717.308,E2 -11717.308} C_VEL
LIN {X 0,Y 390.108,Z 372.885,A -85,B 0,C 180,E1 -11720.482,E2 -11720.482} C_VEL
LIN {X 0,Y 390.084,Z 372.89,A -85,B 0,C 180,E1 -11723.352,E2 -11723.352} C_VEL
LIN {X 0,Y 390.108,Z 372.891,A -85,B 0,C 180,E1 -11726.769,E2 -11726.769} C_VEL
LIN {X 0,Y 390.034,Z 372.898,A -85,B 0,C 180,E1 -11730.301,E2 -11730.301} C_VEL
LIN {X 0,Y 390.064,Z 372.885,A -85,B 0,C 180,E1 -11734.026,E2 -11734.026} C_VEL
LIN {X 0,Y 390.044,Z 372.897,A -85,B 0,C 180,E1 -11737.553,E2 -11737.553} C_VEL
LIN {X 0,Y 390.08,Z 372.897,A -85,B 0,C 180,E1 -11740.827,E2 -11740.827} C_VEL
LIN {X 0,Y 390.102,Z 372.893,A -85,B 0,C 180,E1 -11743.895,E2 -11743.895} C_VEL
LIN {X 0,Y 390.044,Z 372.896,A -85,B 0,C 180,E1 -11747.627,E2 -11747.627} C_VEL
LIN {X 0,Y 390.119,Z 373.007,A -85,B 0,C 180,E1 -11750.231,E2 -11750.231} C_VEL
LIN {X 0,Y 392.028,Z 382.342,A -85,B 0,C 180,E1 -11752.997,E2 -11752.997} C_VEL
LIN {X 0,Y 396.008,Z 392.867,A -85,B 0,C 180,E1 -11753.477,E2 -11753.477} C_VEL
LIN {X 0,Y 398.556,Z 404.141,A -85,B 0,C 180,E1 -11753.86,E2 -11753.86} C_VEL
LIN {X 0,Y 397.076,Z 488.281,A -85,B 0,C 180,E1 -11755.426,E2 -11755.426} C_VEL
LIN {X 0,Y 396.615,Z 501.665,A -85,B 0,C 180,E1 -11755.88,E2 -11755.88} C_VEL
LIN {X 0,Y 396.03,Z 513.722,A -85,B 0,C 180,E1 -11756.488,E2 -11756.488} C_VEL
LIN {X 0,Y 395.192,Z 525.772,A -85,B 0,C 180,E1 -11757.305,E2 -11757.305} C_VEL
LIN {X 0,Y 394.288,Z 536.766,A -85,B 0,C 180,E1 -11758.277,E2 -11758.277} C_VEL
LIN {X 0,Y 393.306,Z 547.074,A -85,B 0,C 180,E1 -11759.416,E2 -11759.416} C_VEL
LIN {X 0,Y 392.287,Z 557.014,A -85,B 0,C 180,E1 -11760.779,E2 -11760.779} C_VEL
LIN {X 0,Y 391.433,Z 565.175,A -85,B 0,C 180,E1 -11762.173,E2 -11762.173} C_VEL
LIN {X 0,Y 390.614,Z 572.793,A -85,B 0,C 180,E1 -11763.785,E2 -11763.785} C_VEL
LIN {X 0,Y 389.947,Z 579.252,A -85,B 0,C 180,E1 -11765.511,E2 -11765.511} C_VEL
LIN {X 0,Y 389.504,Z 583.48,A -85,B 0,C 180,E1 -11766.959,E2 -11766.959} C_VEL
LIN {X 0,Y 389.106,Z 587.574,A -85,B 0,C 180,E1 -11768.824,E2 -11768.824} C_VEL
LIN {X 0,Y 388.88,Z 589.429,A -85,B 0,C 180,E1 -11770.014,E2 -11770.014} C_VEL
LIN {X 0,Y 388.748,Z 590.586,A -85,B 0,C 180,E1 -11771.01,E2 -11771.01} C_VEL
LIN {X 0,Y 388.684,Z 591.423,A -85,B 0,C 180,E1 -11772.099,E2 -11772.099} C_VEL
LIN {X 0,Y 388.643,Z 591.832,A -85,B 0,C 180,E1 -11773.422,E2 -11773.422} C_VEL
LIN {X 0,Y 388.626,Z 591.336,A -85,B 0,C 180,E1 -11775.335,E2 -11775.335} C_VEL
LIN {X 0,Y 388.675,Z 590.441,A -85,B 0,C 180,E1 -11776.405,E2 -11776.405} C_VEL
LIN {X 0,Y 388.773,Z 589.132,A -85,B 0,C 180,E1 -11777.472,E2 -11777.472} C_VEL
LIN {X 0,Y 389.006,Z 586.354,A -85,B 0,C 180,E1 -11779.065,E2 -11779.065} C_VEL
LIN {X 0,Y 389.219,Z 582.55,A -85,B 0,C 180,E1 -11780.648,E2 -11780.648} C_VEL
LIN {X 0,Y 389.621,Z 577.414,A -85,B 0,C 180,E1 -11782.277,E2 -11782.277} C_VEL
LIN {X 0,Y 390.013,Z 571.385,A -85,B 0,C 180,E1 -11783.793,E2 -11783.793} C_VEL
LIN {X 0,Y 390.665,Z 563.616,A -85,B 0,C 180,E1 -11785.357,E2 -11785.357} C_VEL
LIN {X 0,Y 391.455,Z 553.891,A -85,B 0,C 180,E1 -11786.913,E2 -11786.913} C_VEL
LIN {X 0,Y 392.261,Z 543.83,A -85,B 0,C 180,E1 -11788.203,E2 -11788.203} C_VEL
LIN {X 0,Y 393.006,Z 533.568,A -85,B 0,C 180,E1 -11789.257,E2 -11789.257} C_VEL
LIN {X 0,Y 393.716,Z 522.946,A -85,B 0,C 180,E1 -11790.132,E2 -11790.132} C_VEL
LIN {X 0,Y 394.378,Z 510.481,A -85,B 0,C 180,E1 -11790.926,E2 -11790.926} C_VEL
LIN {X 0,Y 394.868,Z 498.03,A -85,B 0,C 180,E1 -11791.498,E2 -11791.498} C_VEL
LIN {X 0,Y 395.147,Z 485.146,A -85,B 0,C 180,E1 -11791.879,E2 -11791.879} C_VEL
LIN {X 0,Y 395.194,Z 483.849,A -85,B 0,C 180,E1 -11791.906,E2 -11791.906} C_VEL
LIN {X 0,Y 394.722,Z 478.046,A -85,B 0,C 180,E1 -11792.047,E2 -11792.047} C_VEL
LIN {X 0,Y 389.389,Z 459.314,A -85,B 0,C 180,E1 -11792.611,E2 -11792.611} C_VEL
LIN {X 0,Y 388.79,Z 453.495,A -85,B 0,C 180,E1 -11792.744,E2 -11792.744} C_VEL
LIN {X 0,Y 389.393,Z 402.837,A -85,B 0,C 180,E1 -11793.685,E2 -11793.685} C_VEL
LIN {X 0,Y 385.882,Z 386.187,A -85,B 0,C 180,E1 -11794.165,E2 -11794.165} C_VEL
LIN {X 0,Y 384.573,Z 381.96,A -85,B 0,C 180,E1 -11794.323,E2 -11794.323} C_VEL
LIN {X 0,Y 383.274,Z 373.745,A -85,B 0,C 180,E1 -11796.647,E2 -11796.647} C_VEL
LIN {X 0,Y 383.137,Z 373.756,A -85,B 0,C 180,E1 -11800.57,E2 -11800.57} C_VEL
LIN {X 0,Y 383.131,Z 373.759,A -85,B 0,C 180,E1 -11803.796,E2 -11803.796} C_VEL
LIN {X 0,Y 383.099,Z 373.766,A -85,B 0,C 180,E1 -11807.454,E2 -11807.454} C_VEL
LIN {X 0,Y 383.035,Z 373.77,A -85,B 0,C 180,E1 -11810.647,E2 -11810.647} C_VEL
LIN {X 0,Y 383.036,Z 373.77,A -85,B 0,C 180,E1 -11813.806,E2 -11813.806} C_VEL
LIN {X 0,Y 383.082,Z 373.763,A -85,B 0,C 180,E1 -11816.122,E2 -11816.122} C_VEL
LIN {X 0,Y 383.044,Z 373.768,A -85,B 0,C 180,E1 -11818.492,E2 -11818.492} C_VEL
LIN {X 0,Y 383.015,Z 373.771,A -85,B 0,C 180,E1 -11822.148,E2 -11822.148} C_VEL
LIN {X 0,Y 383.019,Z 373.773,A -85,B 0,C 180,E1 -11824.667,E2 -11824.667} C_VEL
LIN {X 0,Y 383.002,Z 373.773,A -85,B 0,C 180,E1 -11827.903,E2 -11827.903} C_VEL
LIN {X 0,Y 382.984,Z 373.779,A -85,B 0,C 180,E1 -11831.346,E2 -11831.346} C_VEL
LIN {X 0,Y 382.995,Z 373.774,A -85,B 0,C 180,E1 -11834.302,E2 -11834.302} C_VEL
LIN {X 0,Y 383.008,Z 373.776,A -85,B 0,C 180,E1 -11837.239,E2 -11837.239} C_VEL
LIN {X 0,Y 383.014,Z 373.773,A -85,B 0,C 180,E1 -11840.412,E2 -11840.412} C_VEL
LIN {X 0,Y 383.023,Z 373.77,A -85,B 0,C 180,E1 -11844.044,E2 -11844.044} C_VEL
LIN {X 0,Y 382.982,Z 373.776,A -85,B 0,C 180,E1 -11847.577,E2 -11847.577} C_VEL
LIN {X 0,Y 382.987,Z 373.776,A -85,B 0,C 180,E1 -11850.299,E2 -11850.299} C_VEL
LIN {X 0,Y 383.075,Z 373.764,A -85,B 0,C 180,E1 -11854.02,E2 -11854.02} C_VEL
LIN {X 0,Y 383.002,Z 373.774,A -85,B 0,C 180,E1 -11857.334,E2 -11857.334} C_VEL
LIN {X 0,Y 383.054,Z 373.773,A -85,B 0,C 180,E1 -11860.716,E2 -11860.716} C_VEL
LIN {X 0,Y 383.074,Z 373.765,A -85,B 0,C 180,E1 -11864.026,E2 -11864.026} C_VEL
LIN {X 0,Y 383.129,Z 373.758,A -85,B 0,C 180,E1 -11867.283,E2 -11867.283} C_VEL
LIN {X 0,Y 383.144,Z 373.76,A -85,B 0,C 180,E1 -11870.497,E2 -11870.497} C_VEL
LIN {X 0,Y 383.276,Z 373.739,A -85,B 0,C 180,E1 -11873.683,E2 -11873.683} C_VEL
LIN {X 0,Y 383.38,Z 373.727,A -85,B 0,C 180,E1 -11877.899,E2 -11877.899} C_VEL
LIN {X 0,Y 383.511,Z 373.711,A -85,B 0,C 180,E1 -11880,E2 -11880} C_VEL
LIN {X 0,Y 383.244,Z 373.743,A -85,B 0,C 180,E1 -11883.153,E2 -11883.153} C_VEL
LIN {X 0,Y 383.275,Z 373.744,A -85,B 0,C 180,E1 -11886.316,E2 -11886.316} C_VEL
LIN {X 0,Y 383.143,Z 373.755,A -85,B 0,C 180,E1 -11889.502,E2 -11889.502} C_VEL
LIN {X 0,Y 383.117,Z 373.759,A -85,B 0,C 180,E1 -11893.536,E2 -11893.536} C_VEL
LIN {X 0,Y 383.088,Z 373.762,A -85,B 0,C 180,E1 -11897.455,E2 -11897.455} C_VEL
LIN {X 0,Y 383.021,Z 373.773,A -85,B 0,C 180,E1 -11900.647,E2 -11900.647} C_VEL
LIN {X 0,Y 383.026,Z 373.772,A -85,B 0,C 180,E1 -11903.808,E2 -11903.808} C_VEL
LIN {X 0,Y 383.05,Z 373.767,A -85,B 0,C 180,E1 -11907.302,E2 -11907.302} C_VEL
LIN {X 0,Y 382.98,Z 373.776,A -85,B 0,C 180,E1 -11910.919,E2 -11910.919} C_VEL
LIN {X 0,Y 383.012,Z 373.773,A -85,B 0,C 180,E1 -11914.668,E2 -11914.668} C_VEL
LIN {X 0,Y 382.998,Z 373.778,A -85,B 0,C 180,E1 -11917.905,E2 -11917.905} C_VEL
LIN {X 0,Y 383.042,Z 373.768,A -85,B 0,C 180,E1 -11921.34,E2 -11921.34} C_VEL
LIN {X 0,Y 383.032,Z 373.773,A -85,B 0,C 180,E1 -11924.31,E2 -11924.31} C_VEL
LIN {X 0,Y 383.036,Z 373.769,A -85,B 0,C 180,E1 -11927.245,E2 -11927.245} C_VEL
LIN {X 0,Y 383.019,Z 373.773,A -85,B 0,C 180,E1 -11930.413,E2 -11930.413} C_VEL
LIN {X 0,Y 383.025,Z 373.775,A -85,B 0,C 180,E1 -11934.045,E2 -11934.045} C_VEL
LIN {X 0,Y 383.035,Z 373.775,A -85,B 0,C 180,E1 -11937.854,E2 -11937.854} C_VEL
LIN {X 0,Y 383.119,Z 373.956,A -85,B 0,C 180,E1 -11940.84,E2 -11940.84} C_VEL
LIN {X 0,Y 385.693,Z 386.524,A -85,B 0,C 180,E1 -11943.72,E2 -11943.72} C_VEL
LIN {X 0,Y 386.412,Z 392.286,A -85,B 0,C 180,E1 -11944.985,E2 -11944.985} C_VEL
LIN {X 0,Y 385.249,Z 407.045,A -85,B 0,C 180,E1 -11948.04,E2 -11948.04} C_VEL
LIN {X 0,Y 384.627,Z 415.064,A -85,B 0,C 180,E1 -11949.686,E2 -11949.686} C_VEL
LIN {X 0,Y 389.066,Z 448.118,A -85,B 0,C 180,E1 -11950.518,E2 -11950.518} C_VEL
LIN {X 0,Y 388.03,Z 523.418,A -85,B 0,C 180,E1 -11951.931,E2 -11951.931} C_VEL
LIN {X 0,Y 387.471,Z 536.791,A -85,B 0,C 180,E1 -11952.382,E2 -11952.382} C_VEL
LIN {X 0,Y 386.774,Z 549.613,A -85,B 0,C 180,E1 -11953.031,E2 -11953.031} C_VEL
LIN {X 0,Y 385.883,Z 561.787,A -85,B 0,C 180,E1 -11953.875,E2 -11953.875} C_VEL
LIN {X 0,Y 384.969,Z 573.383,A -85,B 0,C 180,E1 -11954.922,E2 -11954.922} C_VEL
LIN {X 0,Y 384.276,Z 583.499,A -85,B 0,C 180,E1 -11956.068,E2 -11956.068} C_VEL
LIN {X 0,Y 383.508,Z 592.368,A -85,B 0,C 180,E1 -11957.297,E2 -11957.297} C_VEL
LIN {X 0,Y 382.733,Z 601.597,A -85,B 0,C 180,E1 -11958.884,E2 -11958.884} C_VEL
LIN {X 0,Y 382.225,Z 609.028,A -85,B 0,C 180,E1 -11960.475,E2 -11960.475} C_VEL
LIN {X 0,Y 381.905,Z 614.981,A -85,B 0,C 180,E1 -11962.067,E2 -11962.067} C_VEL
LIN {X 0,Y 381.73,Z 620.082,A -85,B 0,C 180,E1 -11963.822,E2 -11963.822} C_VEL
LIN {X 0,Y 381.641,Z 624.16,A -85,B 0,C 180,E1 -11965.776,E2 -11965.776} C_VEL
LIN {X 0,Y 381.601,Z 625.752,A -85,B 0,C 180,E1 -11966.833,E2 -11966.833} C_VEL
LIN {X 0,Y 381.689,Z 626.929,A -85,B 0,C 180,E1 -11967.89,E2 -11967.89} C_VEL
LIN {X 0,Y 381.692,Z 627.654,A -85,B 0,C 180,E1 -11968.945,E2 -11968.945} C_VEL
LIN {X 0,Y 381.69,Z 627.931,A -85,B 0,C 180,E1 -11971.055,E2 -11971.055} C_VEL
LIN {X 0,Y 381.653,Z 627.479,A -85,B 0,C 180,E1 -11972.111,E2 -11972.111} C_VEL
LIN {X 0,Y 381.632,Z 625.302,A -85,B 0,C 180,E1 -11974.224,E2 -11974.224} C_VEL
LIN {X 0,Y 381.695,Z 621.937,A -85,B 0,C 180,E1 -11976.13,E2 -11976.13} C_VEL
LIN {X 0,Y 381.94,Z 617.404,A -85,B 0,C 180,E1 -11977.932,E2 -11977.932} C_VEL
LIN {X 0,Y 382.391,Z 611.166,A -85,B 0,C 180,E1 -11979.788,E2 -11979.788} C_VEL
LIN {X 0,Y 383.018,Z 604.402,A -85,B 0,C 180,E1 -11981.376,E2 -11981.376} C_VEL
LIN {X 0,Y 383.967,Z 596.038,A -85,B 0,C 180,E1 -11982.957,E2 -11982.957} C_VEL
LIN {X 0,Y 384.887,Z 586.41,A -85,B 0,C 180,E1 -11984.415,E2 -11984.415} C_VEL
LIN {X 0,Y 386,Z 575.735,A -85,B 0,C 180,E1 -11985.713,E2 -11985.713} C_VEL
LIN {X 0,Y 387.084,Z 565.038,A -85,B 0,C 180,E1 -11986.752,E2 -11986.752} C_VEL
LIN {X 0,Y 388.211,Z 553.067,A -85,B 0,C 180,E1 -11987.652,E2 -11987.652} C_VEL
LIN {X 0,Y 389.133,Z 540.637,A -85,B 0,C 180,E1 -11988.356,E2 -11988.356} C_VEL
LIN {X 0,Y 389.93,Z 527.724,A -85,B 0,C 180,E1 -11988.862,E2 -11988.862} C_VEL
LIN {X 0,Y 390.285,Z 512.6,A -85,B 0,C 180,E1 -11989.215,E2 -11989.215} C_VEL
LIN {X 0,Y 391.241,Z 446.941,A -85,B 0,C 180,E1 -11990.454,E2 -11990.454} C_VEL
LIN {X 0,Y 388.353,Z 428.208,A -85,B 0,C 180,E1 -11991.014,E2 -11991.014} C_VEL
LIN {X 0,Y 385.698,Z 414.318,A -85,B 0,C 180,E1 -11991.492,E2 -11991.492} C_VEL
LIN {X 0,Y 387.415,Z 396.818,A -85,B 0,C 180,E1 -11995.232,E2 -11995.232} C_VEL
LIN {X 0,Y 387.289,Z 392.957,A -85,B 0,C 180,E1 -11996.107,E2 -11996.107} C_VEL
LIN {X 0,Y 385.228,Z 382.844,A -85,B 0,C 180,E1 -11998.587,E2 -11998.587} C_VEL
LIN {X 0,Y 383.003,Z 373.775,A -85,B 0,C 180,E1 -12000.954,E2 -12000.954} C_VEL
LIN {X 0,Y 383.016,Z 373.777,A -85,B 0,C 180,E1 -12004.339,E2 -12004.339} C_VEL
LIN {X 0,Y 382.996,Z 373.778,A -85,B 0,C 180,E1 -12007.267,E2 -12007.267} C_VEL
LIN {X 0,Y 383.017,Z 373.777,A -85,B 0,C 180,E1 -12009.956,E2 -12009.956} C_VEL
LIN {X 0,Y 383.029,Z 373.768,A -85,B 0,C 180,E1 -12012.782,E2 -12012.782} C_VEL
LIN {X 0,Y 383.036,Z 373.772,A -85,B 0,C 180,E1 -12015.795,E2 -12015.795} C_VEL
LIN {X 0,Y 383.04,Z 373.771,A -85,B 0,C 180,E1 -12018.786,E2 -12018.786} C_VEL
LIN {X 0,Y 382.998,Z 373.776,A -85,B 0,C 180,E1 -12022.095,E2 -12022.095} C_VEL
LIN {X 0,Y 383.012,Z 373.775,A -85,B 0,C 180,E1 -12025.332,E2 -12025.332} C_VEL
LIN {X 0,Y 382.98,Z 373.777,A -85,B 0,C 180,E1 -12029.081,E2 -12029.081} C_VEL
LIN {X 0,Y 383.05,Z 373.767,A -85,B 0,C 180,E1 -12032.698,E2 -12032.698} C_VEL
LIN {X 0,Y 383.045,Z 373.766,A -85,B 0,C 180,E1 -12035.039,E2 -12035.039} C_VEL
LIN {X 0,Y 382.985,Z 373.77,A -85,B 0,C 180,E1 -12038.469,E2 -12038.469} C_VEL
LIN {X 0,Y 383.082,Z 373.761,A -85,B 0,C 180,E1 -12041.828,E2 -12041.828} C_VEL
LIN {X 0,Y 383.105,Z 373.763,A -85,B 0,C 180,E1 -12045.118,E2 -12045.118} C_VEL
LIN {X 0,Y 383.09,Z 373.759,A -85,B 0,C 180,E1 -12048.358,E2 -12048.358} C_VEL
LIN {X 0,Y 383.256,Z 373.735,A -85,B 0,C 180,E1 -12051.976,E2 -12051.976} C_VEL
LIN {X 0,Y 383.192,Z 373.751,A -85,B 0,C 180,E1 -12054.739,E2 -12054.739} C_VEL
LIN {X 0,Y 383.38,Z 373.723,A -85,B 0,C 180,E1 -12057.899,E2 -12057.899} C_VEL
LIN {X 0,Y 383.513,Z 373.711,A -85,B 0,C 180,E1 -12060,E2 -12060} C_VEL
LIN {X 0,Y 383.246,Z 373.739,A -85,B 0,C 180,E1 -12063.154,E2 -12063.154} C_VEL
LIN {X 0,Y 383.255,Z 373.738,A -85,B 0,C 180,E1 -12066.643,E2 -12066.643} C_VEL
LIN {X 0,Y 383.144,Z 373.76,A -85,B 0,C 180,E1 -12069.503,E2 -12069.503} C_VEL
LIN {X 0,Y 383.118,Z 373.763,A -85,B 0,C 180,E1 -12073.537,E2 -12073.537} C_VEL
LIN {X 0,Y 383.089,Z 373.767,A -85,B 0,C 180,E1 -12077.456,E2 -12077.456} C_VEL
LIN {X 0,Y 383.052,Z 373.765,A -85,B 0,C 180,E1 -12080.659,E2 -12080.659} C_VEL
LIN {X 0,Y 383.028,Z 373.766,A -85,B 0,C 180,E1 -12083.808,E2 -12083.808} C_VEL
LIN {X 0,Y 383.051,Z 373.768,A -85,B 0,C 180,E1 -12087.303,E2 -12087.303} C_VEL
LIN {X 0,Y 382.978,Z 373.779,A -85,B 0,C 180,E1 -12090.92,E2 -12090.92} C_VEL
LIN {X 0,Y 383.014,Z 373.763,A -85,B 0,C 180,E1 -12094.669,E2 -12094.669} C_VEL
LIN {X 0,Y 383,Z 373.774,A -85,B 0,C 180,E1 -12097.905,E2 -12097.905} C_VEL
LIN {X 0,Y 383.044,Z 373.768,A -85,B 0,C 180,E1 -12101.34,E2 -12101.34} C_VEL
LIN {X 0,Y 383.035,Z 373.773,A -85,B 0,C 180,E1 -12104.311,E2 -12104.311} C_VEL
LIN {X 0,Y 383.009,Z 373.773,A -85,B 0,C 180,E1 -12107.241,E2 -12107.241} C_VEL
LIN {X 0,Y 383.043,Z 373.856,A -85,B 0,C 180,E1 -12109.832,E2 -12109.832} C_VEL
LIN {X 0,Y 384.94,Z 382.879,A -85,B 0,C 180,E1 -12112.529,E2 -12112.529} C_VEL
LIN {X 0,Y 389.848,Z 395.426,A -85,B 0,C 180,E1 -12113.121,E2 -12113.121} C_VEL
LIN {X 0,Y 392.063,Z 404.98,A -85,B 0,C 180,E1 -12113.46,E2 -12113.46} C_VEL
LIN {X 0,Y 390.487,Z 489.603,A -85,B 0,C 180,E1 -12115.072,E2 -12115.072} C_VEL
LIN {X 0,Y 389.958,Z 502.608,A -85,B 0,C 180,E1 -12115.528,E2 -12115.528} C_VEL
LIN {X 0,Y 389.382,Z 514.158,A -85,B 0,C 180,E1 -12116.126,E2 -12116.126} C_VEL
LIN {X 0,Y 388.478,Z 526.562,A -85,B 0,C 180,E1 -12116.988,E2 -12116.988} C_VEL
LIN {X 0,Y 387.553,Z 537.373,A -85,B 0,C 180,E1 -12117.967,E2 -12117.967} C_VEL
LIN {X 0,Y 386.476,Z 547.957,A -85,B 0,C 180,E1 -12119.163,E2 -12119.163} C_VEL
LIN {X 0,Y 385.447,Z 557.524,A -85,B 0,C 180,E1 -12120.509,E2 -12120.509} C_VEL
LIN {X 0,Y 384.548,Z 565.652,A -85,B 0,C 180,E1 -12121.927,E2 -12121.927} C_VEL
LIN {X 0,Y 383.62,Z 573.61,A -85,B 0,C 180,E1 -12123.654,E2 -12123.654} C_VEL
LIN {X 0,Y 383.028,Z 578.723,A -85,B 0,C 180,E1 -12125.039,E2 -12125.039} C_VEL
LIN {X 0,Y 382.486,Z 583.737,A -85,B 0,C 180,E1 -12126.742,E2 -12126.742} C_VEL
LIN {X 0,Y 382.105,Z 587.44,A -85,B 0,C 180,E1 -12128.417,E2 -12128.417} C_VEL
LIN {X 0,Y 381.869,Z 589.676,A -85,B 0,C 180,E1 -12129.822,E2 -12129.822} C_VEL
LIN {X 0,Y 381.618,Z 591.6,A -85,B 0,C 180,E1 -12131.756,E2 -12131.756} C_VEL
LIN {X 0,Y 381.558,Z 592.159,A -85,B 0,C 180,E1 -12133.297,E2 -12133.297} C_VEL
LIN {X 0,Y 381.521,Z 591.793,A -85,B 0,C 180,E1 -12135.055,E2 -12135.055} C_VEL
LIN {X 0,Y 381.565,Z 591.034,A -85,B 0,C 180,E1 -12136.147,E2 -12136.147} C_VEL
LIN {X 0,Y 381.67,Z 589.573,A -85,B 0,C 180,E1 -12137.407,E2 -12137.407} C_VEL
LIN {X 0,Y 381.934,Z 586.107,A -85,B 0,C 180,E1 -12139.397,E2 -12139.397} C_VEL
LIN {X 0,Y 382.209,Z 582.103,A -85,B 0,C 180,E1 -12141.008,E2 -12141.008} C_VEL
LIN {X 0,Y 382.624,Z 576.637,A -85,B 0,C 180,E1 -12142.693,E2 -12142.693} C_VEL
LIN {X 0,Y 383.104,Z 570.429,A -85,B 0,C 180,E1 -12144.209,E2 -12144.209} C_VEL
LIN {X 0,Y 383.775,Z 562.33,A -85,B 0,C 180,E1 -12145.799,E2 -12145.799} C_VEL
LIN {X 0,Y 384.477,Z 554.064,A -85,B 0,C 180,E1 -12147.119,E2 -12147.119} C_VEL
LIN {X 0,Y 385.327,Z 543.945,A -85,B 0,C 180,E1 -12148.432,E2 -12148.432} C_VEL
LIN {X 0,Y 386.197,Z 532.479,A -85,B 0,C 180,E1 -12149.609,E2 -12149.609} C_VEL
LIN {X 0,Y 387.033,Z 520.286,A -85,B 0,C 180,E1 -12150.587,E2 -12150.587} C_VEL
LIN {X 0,Y 387.616,Z 508.512,A -85,B 0,C 180,E1 -12151.299,E2 -12151.299} C_VEL
LIN {X 0,Y 388.109,Z 495.787,A -85,B 0,C 180,E1 -12151.848,E2 -12151.848} C_VEL
LIN {X 0,Y 388.395,Z 482.631,A -85,B 0,C 180,E1 -12152.205,E2 -12152.205} C_VEL
LIN {X 0,Y 388.79,Z 453.495,A -85,B 0,C 180,E1 -12152.744,E2 -12152.744} C_VEL
LIN {X 0,Y 388.195,Z 447.679,A -85,B 0,C 180,E1 -12152.881,E2 -12152.881} C_VEL
LIN {X 0,Y 382.935,Z 428.951,A -85,B 0,C 180,E1 -12153.471,E2 -12153.471} C_VEL
LIN {X 0,Y 382.484,Z 423.136,A -85,B 0,C 180,E1 -12153.604,E2 -12153.604} C_VEL
LIN {X 0,Y 382.603,Z 403.79,A -85,B 0,C 180,E1 -12153.976,E2 -12153.976} C_VEL
LIN {X 0,Y 379.403,Z 388.474,A -85,B 0,C 180,E1 -12154.426,E2 -12154.426} C_VEL
LIN {X 0,Y 377.432,Z 382.222,A -85,B 0,C 180,E1 -12154.672,E2 -12154.672} C_VEL
LIN {X 0,Y 376.245,Z 374.62,A -85,B 0,C 180,E1 -12156.839,E2 -12156.839} C_VEL
LIN {X 0,Y 376.089,Z 374.635,A -85,B 0,C 180,E1 -12160.77,E2 -12160.77} C_VEL
LIN {X 0,Y 376.07,Z 374.637,A -85,B 0,C 180,E1 -12164.06,E2 -12164.06} C_VEL
LIN {X 0,Y 376.047,Z 374.643,A -85,B 0,C 180,E1 -12167.606,E2 -12167.606} C_VEL
LIN {X 0,Y 375.981,Z 374.649,A -85,B 0,C 180,E1 -12170.831,E2 -12170.831} C_VEL
LIN {X 0,Y 375.997,Z 374.645,A -85,B 0,C 180,E1 -12174.281,E2 -12174.281} C_VEL
LIN {X 0,Y 376.022,Z 374.643,A -85,B 0,C 180,E1 -12176.651,E2 -12176.651} C_VEL
LIN {X 0,Y 375.975,Z 374.654,A -85,B 0,C 180,E1 -12179.078,E2 -12179.078} C_VEL
LIN {X 0,Y 375.953,Z 374.654,A -85,B 0,C 180,E1 -12182.827,E2 -12182.827} C_VEL
LIN {X 0,Y 375.959,Z 374.654,A -85,B 0,C 180,E1 -12185.414,E2 -12185.414} C_VEL
LIN {X 0,Y 375.976,Z 374.648,A -85,B 0,C 180,E1 -12188.27,E2 -12188.27} C_VEL
LIN {X 0,Y 375.934,Z 374.655,A -85,B 0,C 180,E1 -12191.6,E2 -12191.6} C_VEL
LIN {X 0,Y 375.953,Z 374.655,A -85,B 0,C 180,E1 -12195.263,E2 -12195.263} C_VEL
LIN {X 0,Y 375.939,Z 374.658,A -85,B 0,C 180,E1 -12199.132,E2 -12199.132} C_VEL
LIN {X 0,Y 375.963,Z 374.65,A -85,B 0,C 180,E1 -12201.911,E2 -12201.911} C_VEL
LIN {X 0,Y 375.976,Z 374.65,A -85,B 0,C 180,E1 -12205.332,E2 -12205.332} C_VEL
LIN {X 0,Y 375.953,Z 374.653,A -85,B 0,C 180,E1 -12208.437,E2 -12208.437} C_VEL
LIN {X 0,Y 375.978,Z 374.648,A -85,B 0,C 180,E1 -12212.139,E2 -12212.139} C_VEL
LIN {X 0,Y 376.001,Z 374.649,A -85,B 0,C 180,E1 -12214.538,E2 -12214.538} C_VEL
LIN {X 0,Y 375.957,Z 374.651,A -85,B 0,C 180,E1 -12218.045,E2 -12218.045} C_VEL
LIN {X 0,Y 376.002,Z 374.645,A -85,B 0,C 180,E1 -12221.472,E2 -12221.472} C_VEL
LIN {X 0,Y 376.053,Z 374.644,A -85,B 0,C 180,E1 -12224.832,E2 -12224.832} C_VEL
LIN {X 0,Y 376.043,Z 374.641,A -85,B 0,C 180,E1 -12228.136,E2 -12228.136} C_VEL
LIN {X 0,Y 376.212,Z 374.619,A -85,B 0,C 180,E1 -12231.918,E2 -12231.918} C_VEL
LIN {X 0,Y 376.165,Z 374.631,A -85,B 0,C 180,E1 -12234.64,E2 -12234.64} C_VEL
LIN {X 0,Y 376.346,Z 374.603,A -85,B 0,C 180,E1 -12237.859,E2 -12237.859} C_VEL
LIN {X 0,Y 376.48,Z 374.587,A -85,B 0,C 180,E1 -12240,E2 -12240} C_VEL
LIN {X 0,Y 376.182,Z 374.623,A -85,B 0,C 180,E1 -12243.213,E2 -12243.213} C_VEL
LIN {X 0,Y 376.233,Z 374.623,A -85,B 0,C 180,E1 -12246.435,E2 -12246.435} C_VEL
LIN {X 0,Y 376.111,Z 374.632,A -85,B 0,C 180,E1 -12249.681,E2 -12249.681} C_VEL
LIN {X 0,Y 376.081,Z 374.635,A -85,B 0,C 180,E1 -12253.658,E2 -12253.658} C_VEL
LIN {X 0,Y 376.037,Z 374.641,A -85,B 0,C 180,E1 -12257.608,E2 -12257.608} C_VEL
LIN {X 0,Y 375.971,Z 374.65,A -85,B 0,C 180,E1 -12260.832,E2 -12260.832} C_VEL
LIN {X 0,Y 375.987,Z 374.653,A -85,B 0,C 180,E1 -12264.282,E2 -12264.282} C_VEL
LIN {X 0,Y 376.013,Z 374.646,A -85,B 0,C 180,E1 -12266.653,E2 -12266.653} C_VEL
LIN {X 0,Y 375.97,Z 374.649,A -85,B 0,C 180,E1 -12269.079,E2 -12269.079} C_VEL
LIN {X 0,Y 375.945,Z 374.653,A -85,B 0,C 180,E1 -12272.829,E2 -12272.829} C_VEL
LIN {X 0,Y 375.953,Z 374.651,A -85,B 0,C 180,E1 -12275.416,E2 -12275.416} C_VEL
LIN {X 0,Y 375.973,Z 374.653,A -85,B 0,C 180,E1 -12278.272,E2 -12278.272} C_VEL
LIN {X 0,Y 375.985,Z 374.649,A -85,B 0,C 180,E1 -12281.611,E2 -12281.611} C_VEL
LIN {X 0,Y 375.966,Z 374.65,A -85,B 0,C 180,E1 -12285.263,E2 -12285.263} C_VEL
LIN {X 0,Y 375.978,Z 374.648,A -85,B 0,C 180,E1 -12289.139,E2 -12289.139} C_VEL
LIN {X 0,Y 375.966,Z 374.656,A -85,B 0,C 180,E1 -12291.913,E2 -12291.913} C_VEL
LIN {X 0,Y 375.978,Z 374.649,A -85,B 0,C 180,E1 -12295.333,E2 -12295.333} C_VEL
LIN {X 0,Y 375.975,Z 374.649,A -85,B 0,C 180,E1 -12298.44,E2 -12298.44} C_VEL
LIN {X 0,Y 376.058,Z 374.813,A -85,B 0,C 180,E1 -12300.584,E2 -12300.584} C_VEL
LIN {X 0,Y 378.259,Z 385.56,A -85,B 0,C 180,E1 -12303.105,E2 -12303.105} C_VEL
LIN {X 0,Y 379.456,Z 392.995,A -85,B 0,C 180,E1 -12304.787,E2 -12304.787} C_VEL
LIN {X 0,Y 378.255,Z 407.756,A -85,B 0,C 180,E1 -12307.899,E2 -12307.899} C_VEL
LIN {X 0,Y 377.723,Z 414.756,A -85,B 0,C 180,E1 -12309.365,E2 -12309.365} C_VEL
LIN {X 0,Y 382.26,Z 448.432,A -85,B 0,C 180,E1 -12310.232,E2 -12310.232} C_VEL
LIN {X 0,Y 381.172,Z 523.351,A -85,B 0,C 180,E1 -12311.664,E2 -12311.664} C_VEL
LIN {X 0,Y 380.603,Z 536.633,A -85,B 0,C 180,E1 -12312.123,E2 -12312.123} C_VEL
LIN {X 0,Y 379.867,Z 549.406,A -85,B 0,C 180,E1 -12312.782,E2 -12312.782} C_VEL
LIN {X 0,Y 379.022,Z 560.746,A -85,B 0,C 180,E1 -12313.575,E2 -12313.575} C_VEL
LIN {X 0,Y 378.041,Z 572.468,A -85,B 0,C 180,E1 -12314.638,E2 -12314.638} C_VEL
LIN {X 0,Y 377.342,Z 582.289,A -85,B 0,C 180,E1 -12315.756,E2 -12315.756} C_VEL
LIN {X 0,Y 376.512,Z 591.649,A -85,B 0,C 180,E1 -12317.057,E2 -12317.057} C_VEL
LIN {X 0,Y 375.883,Z 599.592,A -85,B 0,C 180,E1 -12318.405,E2 -12318.405} C_VEL
LIN {X 0,Y 375.26,Z 607.329,A -85,B 0,C 180,E1 -12320.024,E2 -12320.024} C_VEL
LIN {X 0,Y 374.848,Z 614.463,A -85,B 0,C 180,E1 -12321.917,E2 -12321.917} C_VEL
LIN {X 0,Y 374.652,Z 619.927,A -85,B 0,C 180,E1 -12323.834,E2 -12323.834} C_VEL
LIN {X 0,Y 374.569,Z 623.739,A -85,B 0,C 180,E1 -12325.696,E2 -12325.696} C_VEL
LIN {X 0,Y 374.589,Z 626.548,A -85,B 0,C 180,E1 -12327.85,E2 -12327.85} C_VEL
LIN {X 0,Y 374.624,Z 627.298,A -85,B 0,C 180,E1 -12328.925,E2 -12328.925} C_VEL
LIN {X 0,Y 374.607,Z 627.645,A -85,B 0,C 180,E1 -12330,E2 -12330} C_VEL
LIN {X 0,Y 374.622,Z 627.605,A -85,B 0,C 180,E1 -12331.075,E2 -12331.075} C_VEL
LIN {X 0,Y 374.552,Z 627.173,A -85,B 0,C 180,E1 -12332.151,E2 -12332.151} C_VEL
LIN {X 0,Y 374.558,Z 625.039,A -85,B 0,C 180,E1 -12334.304,E2 -12334.304} C_VEL
LIN {X 0,Y 374.59,Z 622.05,A -85,B 0,C 180,E1 -12336.077,E2 -12336.077} C_VEL
LIN {X 0,Y 374.877,Z 617.229,A -85,B 0,C 180,E1 -12338.083,E2 -12338.083} C_VEL
LIN {X 0,Y 375.366,Z 611.045,A -85,B 0,C 180,E1 -12339.973,E2 -12339.973} C_VEL
LIN {X 0,Y 376.018,Z 604.328,A -85,B 0,C 180,E1 -12341.591,E2 -12341.591} C_VEL
LIN {X 0,Y 377.042,Z 596.024,A -85,B 0,C 180,E1 -12343.199,E2 -12343.199} C_VEL
LIN {X 0,Y 377.999,Z 586.49,A -85,B 0,C 180,E1 -12344.684,E2 -12344.684} C_VEL
LIN {X 0,Y 379.162,Z 575.899,A -85,B 0,C 180,E1 -12346.004,E2 -12346.004} C_VEL
LIN {X 0,Y 380.3,Z 565.329,A -85,B 0,C 180,E1 -12347.06,E2 -12347.06} C_VEL
LIN {X 0,Y 381.482,Z 553.586,A -85,B 0,C 180,E1 -12347.973,E2 -12347.973} C_VEL
LIN {X 0,Y 382.55,Z 540.145,A -85,B 0,C 180,E1 -12348.753,E2 -12348.753} C_VEL
LIN {X 0,Y 383.336,Z 527.157,A -85,B 0,C 180,E1 -12349.269,E2 -12349.269} C_VEL
LIN {X 0,Y 383.744,Z 511.773,A -85,B 0,C 180,E1 -12349.628,E2 -12349.628} C_VEL
LIN {X 0,Y 384.836,Z 448.572,A -85,B 0,C 180,E1 -12350.836,E2 -12350.836} C_VEL
LIN {X 0,Y 382.116,Z 430.547,A -85,B 0,C 180,E1 -12351.386,E2 -12351.386} C_VEL
LIN {X 0,Y 378.95,Z 413.914,A -85,B 0,C 180,E1 -12351.982,E2 -12351.982} C_VEL
LIN {X 0,Y 380.683,Z 396.847,A -85,B 0,C 180,E1 -12355.711,E2 -12355.711} C_VEL
LIN {X 0,Y 379.405,Z 389.176,A -85,B 0,C 180,E1 -12357.586,E2 -12357.586} C_VEL
LIN {X 0,Y 376.463,Z 376.719,A -85,B 0,C 180,E1 -12360.823,E2 -12360.823} C_VEL
LIN {X 0,Y 375.993,Z 374.648,A -85,B 0,C 180,E1 -12361.444,E2 -12361.444} C_VEL
LIN {X 0,Y 375.956,Z 374.654,A -85,B 0,C 180,E1 -12365.415,E2 -12365.415} C_VEL
LIN {X 0,Y 375.976,Z 374.646,A -85,B 0,C 180,E1 -12368.271,E2 -12368.271} C_VEL
LIN {X 0,Y 375.957,Z 374.647,A -85,B 0,C 180,E1 -12371.605,E2 -12371.605} C_VEL
LIN {X 0,Y 375.976,Z 374.65,A -85,B 0,C 180,E1 -12375.26,E2 -12375.26} C_VEL
LIN {X 0,Y 375.985,Z 374.651,A -85,B 0,C 180,E1 -12378.389,E2 -12378.389} C_VEL
LIN {X 0,Y 375.963,Z 374.655,A -85,B 0,C 180,E1 -12381.911,E2 -12381.911} C_VEL
LIN {X 0,Y 375.974,Z 374.652,A -85,B 0,C 180,E1 -12385.332,E2 -12385.332} C_VEL
LIN {X 0,Y 375.954,Z 374.652,A -85,B 0,C 180,E1 -12388.438,E2 -12388.438} C_VEL
LIN {X 0,Y 375.996,Z 374.648,A -85,B 0,C 180,E1 -12392.141,E2 -12392.141} C_VEL
LIN {X 0,Y 375.999,Z 374.643,A -85,B 0,C 180,E1 -12394.539,E2 -12394.539} C_VEL
LIN {X 0,Y 375.955,Z 374.646,A -85,B 0,C 180,E1 -12398.045,E2 -12398.045} C_VEL
LIN {X 0,Y 376.016,Z 374.646,A -85,B 0,C 180,E1 -12401.474,E2 -12401.474} C_VEL
LIN {X 0,Y 376.053,Z 374.64,A -85,B 0,C 180,E1 -12404.833,E2 -12404.833} C_VEL
LIN {X 0,Y 376.042,Z 374.638,A -85,B 0,C 180,E1 -12408.137,E2 -12408.137} C_VEL
LIN {X 0,Y 376.211,Z 374.613,A -85,B 0,C 180,E1 -12411.919,E2 -12411.919} C_VEL
LIN {X 0,Y 376.164,Z 374.626,A -85,B 0,C 180,E1 -12414.64,E2 -12414.64} C_VEL
LIN {X 0,Y 376.346,Z 374.599,A -85,B 0,C 180,E1 -12417.86,E2 -12417.86} C_VEL
LIN {X 0,Y 376.482,Z 374.587,A -85,B 0,C 180,E1 -12420,E2 -12420} C_VEL
LIN {X 0,Y 376.184,Z 374.619,A -85,B 0,C 180,E1 -12423.213,E2 -12423.213} C_VEL
LIN {X 0,Y 376.22,Z 374.615,A -85,B 0,C 180,E1 -12426.632,E2 -12426.632} C_VEL
LIN {X 0,Y 376.112,Z 374.634,A -85,B 0,C 180,E1 -12429.682,E2 -12429.682} C_VEL
LIN {X 0,Y 376.082,Z 374.638,A -85,B 0,C 180,E1 -12433.658,E2 -12433.658} C_VEL
LIN {X 0,Y 376.038,Z 374.644,A -85,B 0,C 180,E1 -12437.608,E2 -12437.608} C_VEL
LIN {X 0,Y 376.001,Z 374.644,A -85,B 0,C 180,E1 -12440.844,E2 -12440.844} C_VEL
LIN {X 0,Y 375.988,Z 374.643,A -85,B 0,C 180,E1 -12444.282,E2 -12444.282} C_VEL
LIN {X 0,Y 376.014,Z 374.647,A -85,B 0,C 180,E1 -12446.653,E2 -12446.653} C_VEL
LIN {X 0,Y 375.96,Z 374.651,A -85,B 0,C 180,E1 -12450.314,E2 -12450.314} C_VEL
LIN {X 0,Y 375.956,Z 374.641,A -85,B 0,C 180,E1 -12454.112,E2 -12454.112} C_VEL
LIN {X 0,Y 375.952,Z 374.659,A -85,B 0,C 180,E1 -12456.742,E2 -12456.742} C_VEL
LIN {X 0,Y 375.996,Z 374.647,A -85,B 0,C 180,E1 -12459.974,E2 -12459.974} C_VEL
LIN {X 0,Y 375.988,Z 374.65,A -85,B 0,C 180,E1 -12463.2,E2 -12463.2} C_VEL
LIN {X 0,Y 375.936,Z 374.656,A -85,B 0,C 180,E1 -12466.811,E2 -12466.811} C_VEL
LIN {X 0,Y 376.007,Z 374.805,A -85,B 0,C 180,E1 -12469.443,E2 -12469.443} C_VEL
LIN {X 0,Y 377.826,Z 383.261,A -85,B 0,C 180,E1 -12472.023,E2 -12472.023} C_VEL
LIN {X 0,Y 383.551,Z 397.466,A -85,B 0,C 180,E1 -12472.729,E2 -12472.729} C_VEL
LIN {X 0,Y 385.604,Z 406.352,A -85,B 0,C 180,E1 -12473.053,E2 -12473.053} C_VEL
LIN {X 0,Y 383.962,Z 489.911,A -85,B 0,C 180,E1 -12474.671,E2 -12474.671} C_VEL
LIN {X 0,Y 383.394,Z 503.323,A -85,B 0,C 180,E1 -12475.152,E2 -12475.152} C_VEL
LIN {X 0,Y 382.72,Z 515.29,A -85,B 0,C 180,E1 -12475.789,E2 -12475.789} C_VEL
LIN {X 0,Y 381.802,Z 527.148,A -85,B 0,C 180,E1 -12476.639,E2 -12476.639} C_VEL
LIN {X 0,Y 380.829,Z 538.002,A -85,B 0,C 180,E1 -12477.645,E2 -12477.645} C_VEL
LIN {X 0,Y 379.637,Z 549.106,A -85,B 0,C 180,E1 -12478.934,E2 -12478.934} C_VEL
LIN {X 0,Y 378.636,Z 557.878,A -85,B 0,C 180,E1 -12480.204,E2 -12480.204} C_VEL
LIN {X 0,Y 377.655,Z 566.126,A -85,B 0,C 180,E1 -12481.671,E2 -12481.671} C_VEL
LIN {X 0,Y 376.681,Z 573.94,A -85,B 0,C 180,E1 -12483.399,E2 -12483.399} C_VEL
LIN {X 0,Y 375.965,Z 580.1,A -85,B 0,C 180,E1 -12485.128,E2 -12485.128} C_VEL
LIN {X 0,Y 375.39,Z 584.827,A -85,B 0,C 180,E1 -12486.849,E2 -12486.849} C_VEL
LIN {X 0,Y 375.116,Z 587.278,A -85,B 0,C 180,E1 -12487.994,E2 -12487.994} C_VEL
LIN {X 0,Y 374.821,Z 589.956,A -85,B 0,C 180,E1 -12489.64,E2 -12489.64} C_VEL
LIN {X 0,Y 374.549,Z 591.754,A -85,B 0,C 180,E1 -12491.399,E2 -12491.399} C_VEL
LIN {X 0,Y 374.473,Z 592.487,A -85,B 0,C 180,E1 -12493.169,E2 -12493.169} C_VEL
LIN {X 0,Y 374.426,Z 592.243,A -85,B 0,C 180,E1 -12494.765,E2 -12494.765} C_VEL
LIN {X 0,Y 374.456,Z 591.56,A -85,B 0,C 180,E1 -12495.878,E2 -12495.878} C_VEL
LIN {X 0,Y 374.581,Z 590.017,A -85,B 0,C 180,E1 -12497.33,E2 -12497.33} C_VEL
LIN {X 0,Y 374.832,Z 586.925,A -85,B 0,C 180,E1 -12499.193,E2 -12499.193} C_VEL
LIN {X 0,Y 375.086,Z 583.084,A -85,B 0,C 180,E1 -12500.836,E2 -12500.836} C_VEL
LIN {X 0,Y 375.54,Z 577.356,A -85,B 0,C 180,E1 -12502.691,E2 -12502.691} C_VEL
LIN {X 0,Y 376.088,Z 570.63,A -85,B 0,C 180,E1 -12504.37,E2 -12504.37} C_VEL
LIN {X 0,Y 376.79,Z 562.504,A -85,B 0,C 180,E1 -12505.989,E2 -12505.989} C_VEL
LIN {X 0,Y 377.522,Z 554.206,A -85,B 0,C 180,E1 -12507.333,E2 -12507.333} C_VEL
LIN {X 0,Y 378.424,Z 544.02,A -85,B 0,C 180,E1 -12508.67,E2 -12508.67} C_VEL
LIN {X 0,Y 379.31,Z 532.507,A -85,B 0,C 180,E1 -12509.867,E2 -12509.867} C_VEL
LIN {X 0,Y 380.118,Z 521.078,A -85,B 0,C 180,E1 -12510.801,E2 -12510.801} C_VEL
LIN {X 0,Y 380.719,Z 509.59,A -85,B 0,C 180,E1 -12511.521,E2 -12511.521} C_VEL
LIN {X 0,Y 381.246,Z 496.275,A -85,B 0,C 180,E1 -12512.113,E2 -12512.113} C_VEL
LIN {X 0,Y 381.547,Z 483.297,A -85,B 0,C 180,E1 -12512.474,E2 -12512.474} C_VEL
LIN {X 0,Y 382.484,Z 423.136,A -85,B 0,C 180,E1 -12513.604,E2 -12513.604} C_VEL
LIN {X 0,Y 382.017,Z 417.305,A -85,B 0,C 180,E1 -12513.739,E2 -12513.739} C_VEL
LIN {X 0,Y 380.51,Z 411.667,A -85,B 0,C 180,E1 -12513.919,E2 -12513.919} C_VEL
LIN {X 0,Y 376.117,Z 400.737,A -85,B 0,C 180,E1 -12514.338,E2 -12514.338} C_VEL
LIN {X 0,Y 373.536,Z 393.273,A -85,B 0,C 180,E1 -12514.61,E2 -12514.61} C_VEL
LIN {X 0,Y 370.356,Z 382.598,A -85,B 0,C 180,E1 -12515.001,E2 -12515.001} C_VEL
LIN {X 0,Y 369.204,Z 375.497,A -85,B 0,C 180,E1 -12517.039,E2 -12517.039} C_VEL
LIN {X 0,Y 369.027,Z 375.516,A -85,B 0,C 180,E1 -12520.979,E2 -12520.979} C_VEL
LIN {X 0,Y 369.02,Z 375.515,A -85,B 0,C 180,E1 -12524.334,E2 -12524.334} C_VEL
LIN {X 0,Y 369.005,Z 375.519,A -85,B 0,C 180,E1 -12527.768,E2 -12527.768} C_VEL
LIN {X 0,Y 368.933,Z 375.531,A -85,B 0,C 180,E1 -12531.219,E2 -12531.219} C_VEL
LIN {X 0,Y 368.961,Z 375.524,A -85,B 0,C 180,E1 -12534.775,E2 -12534.775} C_VEL
LIN {X 0,Y 368.971,Z 375.527,A -85,B 0,C 180,E1 -12537.202,E2 -12537.202} C_VEL
LIN {X 0,Y 368.923,Z 375.528,A -85,B 0,C 180,E1 -12539.689,E2 -12539.689} C_VEL
LIN {X 0,Y 368.9,Z 375.532,A -85,B 0,C 180,E1 -12543.537,E2 -12543.537} C_VEL
LIN {X 0,Y 368.903,Z 375.533,A -85,B 0,C 180,E1 -12546.855,E2 -12546.855} C_VEL
LIN {X 0,Y 368.911,Z 375.529,A -85,B 0,C 180,E1 -12550.369,E2 -12550.369} C_VEL
LIN {X 0,Y 368.882,Z 375.533,A -85,B 0,C 180,E1 -12553.615,E2 -12553.615} C_VEL
LIN {X 0,Y 368.884,Z 375.535,A -85,B 0,C 180,E1 -12556.695,E2 -12556.695} C_VEL
LIN {X 0,Y 368.91,Z 375.529,A -85,B 0,C 180,E1 -12559.642,E2 -12559.642} C_VEL
LIN {X 0,Y 368.9,Z 375.534,A -85,B 0,C 180,E1 -12563.143,E2 -12563.143} C_VEL
LIN {X 0,Y 368.892,Z 375.533,A -85,B 0,C 180,E1 -12566.461,E2 -12566.461} C_VEL
LIN {X 0,Y 368.925,Z 375.531,A -85,B 0,C 180,E1 -12569.046,E2 -12569.046} C_VEL
LIN {X 0,Y 368.958,Z 375.529,A -85,B 0,C 180,E1 -12572.796,E2 -12572.796} C_VEL
LIN {X 0,Y 368.939,Z 375.525,A -85,B 0,C 180,E1 -12576.112,E2 -12576.112} C_VEL
LIN {X 0,Y 368.93,Z 375.526,A -85,B 0,C 180,E1 -12579.946,E2 -12579.946} C_VEL
LIN {X 0,Y 368.969,Z 375.522,A -85,B 0,C 180,E1 -12583.398,E2 -12583.398} C_VEL
LIN {X 0,Y 369.051,Z 375.516,A -85,B 0,C 180,E1 -12586.79,E2 -12586.79} C_VEL
LIN {X 0,Y 369.06,Z 375.511,A -85,B 0,C 180,E1 -12590.131,E2 -12590.131} C_VEL
LIN {X 0,Y 369.194,Z 375.493,A -85,B 0,C 180,E1 -12593.441,E2 -12593.441} C_VEL
LIN {X 0,Y 369.311,Z 375.479,A -85,B 0,C 180,E1 -12597.819,E2 -12597.819} C_VEL
LIN {X 0,Y 369.45,Z 375.463,A -85,B 0,C 180,E1 -12600,E2 -12600} C_VEL
LIN {X 0,Y 369.311,Z 375.481,A -85,B 0,C 180,E1 -12602.181,E2 -12602.181} C_VEL
LIN {X 0,Y 369.193,Z 375.499,A -85,B 0,C 180,E1 -12606.558,E2 -12606.558} C_VEL
LIN {X 0,Y 369.06,Z 375.511,A -85,B 0,C 180,E1 -12609.868,E2 -12609.868} C_VEL
LIN {X 0,Y 369.029,Z 375.514,A -85,B 0,C 180,E1 -12613.772,E2 -12613.772} C_VEL
LIN {X 0,Y 368.994,Z 375.519,A -85,B 0,C 180,E1 -12617.769,E2 -12617.769} C_VEL
LIN {X 0,Y 368.922,Z 375.527,A -85,B 0,C 180,E1 -12621.22,E2 -12621.22} C_VEL
LIN {X 0,Y 368.95,Z 375.525,A -85,B 0,C 180,E1 -12624.776,E2 -12624.776} C_VEL
LIN {X 0,Y 368.98,Z 375.524,A -85,B 0,C 180,E1 -12628.436,E2 -12628.436} C_VEL
LIN {X 0,Y 368.894,Z 375.536,A -85,B 0,C 180,E1 -12632.238,E2 -12632.238} C_VEL
LIN {X 0,Y 368.924,Z 375.527,A -85,B 0,C 180,E1 -12635.002,E2 -12635.002} C_VEL
LIN {X 0,Y 368.908,Z 375.53,A -85,B 0,C 180,E1 -12638.642,E2 -12638.642} C_VEL
LIN {X 0,Y 368.947,Z 375.53,A -85,B 0,C 180,E1 -12642.022,E2 -12642.022} C_VEL
LIN {X 0,Y 368.92,Z 375.527,A -85,B 0,C 180,E1 -12645.183,E2 -12645.183} C_VEL
LIN {X 0,Y 368.907,Z 375.533,A -85,B 0,C 180,E1 -12648.182,E2 -12648.182} C_VEL
LIN {X 0,Y 368.911,Z 375.529,A -85,B 0,C 180,E1 -12651.359,E2 -12651.359} C_VEL
LIN {X 0,Y 368.935,Z 375.526,A -85,B 0,C 180,E1 -12655.147,E2 -12655.147} C_VEL
LIN {X 0,Y 368.928,Z 375.526,A -85,B 0,C 180,E1 -12659.047,E2 -12659.047} C_VEL
LIN {X 0,Y 368.96,Z 375.645,A -85,B 0,C 180,E1 -12660.314,E2 -12660.314} C_VEL
LIN {X 0,Y 371.281,Z 386.79,A -85,B 0,C 180,E1 -12662.981,E2 -12662.981} C_VEL
LIN {X 0,Y 372.478,Z 394.15,A -85,B 0,C 180,E1 -12664.682,E2 -12664.682} C_VEL
LIN {X 0,Y 371.277,Z 408.443,A -85,B 0,C 180,E1 -12667.754,E2 -12667.754} C_VEL
LIN {X 0,Y 370.795,Z 414.352,A -85,B 0,C 180,E1 -12669.017,E2 -12669.017} C_VEL
LIN {X 0,Y 375.455,Z 448.669,A -85,B 0,C 180,E1 -12669.933,E2 -12669.933} C_VEL
LIN {X 0,Y 374.318,Z 523.275,A -85,B 0,C 180,E1 -12671.387,E2 -12671.387} C_VEL
LIN {X 0,Y 373.746,Z 536.475,A -85,B 0,C 180,E1 -12671.854,E2 -12671.854} C_VEL
LIN {X 0,Y 372.985,Z 549.203,A -85,B 0,C 180,E1 -12672.525,E2 -12672.525} C_VEL
LIN {X 0,Y 372.027,Z 561.3,A -85,B 0,C 180,E1 -12673.398,E2 -12673.398} C_VEL
LIN {X 0,Y 371.034,Z 572.862,A -85,B 0,C 180,E1 -12674.482,E2 -12674.482} C_VEL
LIN {X 0,Y 370.268,Z 583.303,A -85,B 0,C 180,E1 -12675.715,E2 -12675.715} C_VEL
LIN {X 0,Y 369.419,Z 592.645,A -85,B 0,C 180,E1 -12677.083,E2 -12677.083} C_VEL
LIN {X 0,Y 368.598,Z 601.71,A -85,B 0,C 180,E1 -12678.73,E2 -12678.73} C_VEL
LIN {X 0,Y 368.075,Z 609.009,A -85,B 0,C 180,E1 -12680.383,E2 -12680.383} C_VEL
LIN {X 0,Y 367.783,Z 613.927,A -85,B 0,C 180,E1 -12681.76,E2 -12681.76} C_VEL
LIN {X 0,Y 367.625,Z 618.701,A -85,B 0,C 180,E1 -12683.414,E2 -12683.414} C_VEL
LIN {X 0,Y 367.492,Z 622.332,A -85,B 0,C 180,E1 -12685.063,E2 -12685.063} C_VEL
LIN {X 0,Y 367.426,Z 624.933,A -85,B 0,C 180,E1 -12686.71,E2 -12686.71} C_VEL
LIN {X 0,Y 367.49,Z 626.156,A -85,B 0,C 180,E1 -12687.808,E2 -12687.808} C_VEL
LIN {X 0,Y 367.558,Z 626.938,A -85,B 0,C 180,E1 -12688.904,E2 -12688.904} C_VEL
LIN {X 0,Y 367.541,Z 627.303,A -85,B 0,C 180,E1 -12690,E2 -12690} C_VEL
LIN {X 0,Y 367.536,Z 627.279,A -85,B 0,C 180,E1 -12691.096,E2 -12691.096} C_VEL
LIN {X 0,Y 367.452,Z 626.864,A -85,B 0,C 180,E1 -12692.192,E2 -12692.192} C_VEL
LIN {X 0,Y 367.408,Z 626.033,A -85,B 0,C 180,E1 -12693.29,E2 -12693.29} C_VEL
LIN {X 0,Y 367.462,Z 624.781,A -85,B 0,C 180,E1 -12694.387,E2 -12694.387} C_VEL
LIN {X 0,Y 367.516,Z 622.077,A -85,B 0,C 180,E1 -12696.068,E2 -12696.068} C_VEL
LIN {X 0,Y 367.706,Z 618.49,A -85,B 0,C 180,E1 -12697.689,E2 -12697.689} C_VEL
LIN {X 0,Y 368.086,Z 613.747,A -85,B 0,C 180,E1 -12699.34,E2 -12699.34} C_VEL
LIN {X 0,Y 368.77,Z 606.644,A -85,B 0,C 180,E1 -12701.265,E2 -12701.265} C_VEL
LIN {X 0,Y 369.75,Z 598.982,A -85,B 0,C 180,E1 -12702.905,E2 -12702.905} C_VEL
LIN {X 0,Y 370.816,Z 589.535,A -85,B 0,C 180,E1 -12704.521,E2 -12704.521} C_VEL
LIN {X 0,Y 371.929,Z 579.535,A -85,B 0,C 180,E1 -12705.902,E2 -12705.902} C_VEL
LIN {X 0,Y 373.251,Z 568.508,A -85,B 0,C 180,E1 -12707.109,E2 -12707.109} C_VEL
LIN {X 0,Y 374.423,Z 557.737,A -85,B 0,C 180,E1 -12708.041,E2 -12708.041} C_VEL
LIN {X 0,Y 375.533,Z 545.902,A -85,B 0,C 180,E1 -12708.834,E2 -12708.834} C_VEL
LIN {X 0,Y 376.415,Z 533.179,A -85,B 0,C 180,E1 -12709.46,E2 -12709.46} C_VEL
LIN {X 0,Y 377.033,Z 520.094,A -85,B 0,C 180,E1 -12709.871,E2 -12709.871} C_VEL
LIN {X 0,Y 378.29,Z 448.84,A -85,B 0,C 180,E1 -12711.271,E2 -12711.271} C_VEL
LIN {X 0,Y 375.49,Z 430.847,A -85,B 0,C 180,E1 -12711.841,E2 -12711.841} C_VEL
LIN {X 0,Y 372.194,Z 413.663,A -85,B 0,C 180,E1 -12712.455,E2 -12712.455} C_VEL
LIN {X 0,Y 373.821,Z 398.156,A -85,B 0,C 180,E1 -12715.919,E2 -12715.919} C_VEL
LIN {X 0,Y 372.521,Z 390.762,A -85,B 0,C 180,E1 -12717.769,E2 -12717.769} C_VEL
LIN {X 0,Y 369.786,Z 379.08,A -85,B 0,C 180,E1 -12720.873,E2 -12720.873} C_VEL
LIN {X 0,Y 368.931,Z 375.53,A -85,B 0,C 180,E1 -12721.881,E2 -12721.881} C_VEL
LIN {X 0,Y 368.927,Z 375.529,A -85,B 0,C 180,E1 -12725.001,E2 -12725.001} C_VEL
LIN {X 0,Y 368.911,Z 375.525,A -85,B 0,C 180,E1 -12728.641,E2 -12728.641} C_VEL
LIN {X 0,Y 368.907,Z 375.524,A -85,B 0,C 180,E1 -12731.818,E2 -12731.818} C_VEL
LIN {X 0,Y 368.951,Z 375.525,A -85,B 0,C 180,E1 -12735.187,E2 -12735.187} C_VEL
LIN {X 0,Y 368.937,Z 375.529,A -85,B 0,C 180,E1 -12738.185,E2 -12738.185} C_VEL
LIN {X 0,Y 368.908,Z 375.531,A -85,B 0,C 180,E1 -12741.358,E2 -12741.358} C_VEL
LIN {X 0,Y 368.931,Z 375.528,A -85,B 0,C 180,E1 -12745.146,E2 -12745.146} C_VEL
LIN {X 0,Y 368.923,Z 375.528,A -85,B 0,C 180,E1 -12749.046,E2 -12749.046} C_VEL
LIN {X 0,Y 368.98,Z 375.522,A -85,B 0,C 180,E1 -12751.564,E2 -12751.564} C_VEL
LIN {X 0,Y 368.95,Z 375.523,A -85,B 0,C 180,E1 -12755.224,E2 -12755.224} C_VEL
LIN {X 0,Y 368.93,Z 375.522,A -85,B 0,C 180,E1 -12758.973,E2 -12758.973} C_VEL
LIN {X 0,Y 368.983,Z 375.514,A -85,B 0,C 180,E1 -12762.257,E2 -12762.257} C_VEL
LIN {X 0,Y 369.029,Z 375.513,A -85,B 0,C 180,E1 -12766.228,E2 -12766.228} C_VEL
LIN {X 0,Y 369.06,Z 375.512,A -85,B 0,C 180,E1 -12770.132,E2 -12770.132} C_VEL
LIN {X 0,Y 369.154,Z 375.49,A -85,B 0,C 180,E1 -12772.342,E2 -12772.342} C_VEL
LIN {X 0,Y 369.136,Z 375.501,A -85,B 0,C 180,E1 -12774.538,E2 -12774.538} C_VEL
LIN {X 0,Y 369.311,Z 375.474,A -85,B 0,C 180,E1 -12777.819,E2 -12777.819} C_VEL
LIN {X 0,Y 369.452,Z 375.463,A -85,B 0,C 180,E1 -12780,E2 -12780} C_VEL
LIN {X 0,Y 369.312,Z 375.471,A -85,B 0,C 180,E1 -12782.181,E2 -12782.181} C_VEL
LIN {X 0,Y 369.19,Z 375.492,A -85,B 0,C 180,E1 -12786.617,E2 -12786.617} C_VEL
LIN {X 0,Y 369.06,Z 375.512,A -85,B 0,C 180,E1 -12789.869,E2 -12789.869} C_VEL
LIN {X 0,Y 369.03,Z 375.516,A -85,B 0,C 180,E1 -12793.773,E2 -12793.773} C_VEL
LIN {X 0,Y 368.995,Z 375.52,A -85,B 0,C 180,E1 -12797.769,E2 -12797.769} C_VEL
LIN {X 0,Y 368.959,Z 375.524,A -85,B 0,C 180,E1 -12801.218,E2 -12801.218} C_VEL
LIN {X 0,Y 368.952,Z 375.523,A -85,B 0,C 180,E1 -12804.776,E2 -12804.776} C_VEL
LIN {X 0,Y 368.958,Z 375.523,A -85,B 0,C 180,E1 -12807.204,E2 -12807.204} C_VEL
LIN {X 0,Y 368.925,Z 375.53,A -85,B 0,C 180,E1 -12810.954,E2 -12810.954} C_VEL
LIN {X 0,Y 368.925,Z 375.519,A -85,B 0,C 180,E1 -12815.002,E2 -12815.002} C_VEL
LIN {X 0,Y 368.911,Z 375.534,A -85,B 0,C 180,E1 -12818.642,E2 -12818.642} C_VEL
LIN {X 0,Y 368.94,Z 375.521,A -85,B 0,C 180,E1 -12822.021,E2 -12822.021} C_VEL
LIN {X 0,Y 368.923,Z 375.526,A -85,B 0,C 180,E1 -12825.184,E2 -12825.184} C_VEL
LIN {X 0,Y 368.955,Z 375.713,A -85,B 0,C 180,E1 -12829.018,E2 -12829.018} C_VEL
LIN {X 0,Y 370.656,Z 383.482,A -85,B 0,C 180,E1 -12831.484,E2 -12831.484} C_VEL
LIN {X 0,Y 377.496,Z 400.185,A -85,B 0,C 180,E1 -12832.354,E2 -12832.354} C_VEL
LIN {X 0,Y 379.141,Z 407.271,A -85,B 0,C 180,E1 -12832.62,E2 -12832.62} C_VEL
LIN {X 0,Y 377.434,Z 490.225,A -85,B 0,C 180,E1 -12834.253,E2 -12834.253} C_VEL
LIN {X 0,Y 376.839,Z 503.459,A -85,B 0,C 180,E1 -12834.733,E2 -12834.733} C_VEL
LIN {X 0,Y 376.092,Z 516.397,A -85,B 0,C 180,E1 -12835.438,E2 -12835.438} C_VEL
LIN {X 0,Y 375.154,Z 527.907,A -85,B 0,C 180,E1 -12836.291,E2 -12836.291} C_VEL
LIN {X 0,Y 374.055,Z 539.315,A -85,B 0,C 180,E1 -12837.379,E2 -12837.379} C_VEL
LIN {X 0,Y 372.873,Z 549.716,A -85,B 0,C 180,E1 -12838.623,E2 -12838.623} C_VEL
LIN {X 0,Y 371.803,Z 558.581,A -85,B 0,C 180,E1 -12839.941,E2 -12839.941} C_VEL
LIN {X 0,Y 370.794,Z 566.63,A -85,B 0,C 180,E1 -12841.408,E2 -12841.408} C_VEL
LIN {X 0,Y 369.923,Z 573.23,A -85,B 0,C 180,E1 -12842.874,E2 -12842.874} C_VEL
LIN {X 0,Y 369.095,Z 579.59,A -85,B 0,C 180,E1 -12844.633,E2 -12844.633} C_VEL
LIN {X 0,Y 368.48,Z 584.53,A -85,B 0,C 180,E1 -12846.389,E2 -12846.389} C_VEL
LIN {X 0,Y 368.013,Z 588.223,A -85,B 0,C 180,E1 -12848.137,E2 -12848.137} C_VEL
LIN {X 0,Y 367.687,Z 590.787,A -85,B 0,C 180,E1 -12849.876,E2 -12849.876} C_VEL
LIN {X 0,Y 367.496,Z 591.908,A -85,B 0,C 180,E1 -12851.028,E2 -12851.028} C_VEL
LIN {X 0,Y 367.392,Z 592.816,A -85,B 0,C 180,E1 -12853.035,E2 -12853.035} C_VEL
LIN {X 0,Y 367.355,Z 592.692,A -85,B 0,C 180,E1 -12854.465,E2 -12854.465} C_VEL
LIN {X 0,Y 367.36,Z 592.082,A -85,B 0,C 180,E1 -12855.6,E2 -12855.6} C_VEL
LIN {X 0,Y 367.494,Z 590.463,A -85,B 0,C 180,E1 -12857.25,E2 -12857.25} C_VEL
LIN {X 0,Y 367.794,Z 586.657,A -85,B 0,C 180,E1 -12859.541,E2 -12859.541} C_VEL
LIN {X 0,Y 368.108,Z 582.61,A -85,B 0,C 180,E1 -12861.215,E2 -12861.215} C_VEL
LIN {X 0,Y 368.543,Z 577.289,A -85,B 0,C 180,E1 -12862.908,E2 -12862.908} C_VEL
LIN {X 0,Y 369.075,Z 570.831,A -85,B 0,C 180,E1 -12864.537,E2 -12864.537} C_VEL
LIN {X 0,Y 369.804,Z 562.679,A -85,B 0,C 180,E1 -12866.186,E2 -12866.186} C_VEL
LIN {X 0,Y 370.569,Z 554.349,A -85,B 0,C 180,E1 -12867.554,E2 -12867.554} C_VEL
LIN {X 0,Y 371.511,Z 544.101,A -85,B 0,C 180,E1 -12868.916,E2 -12868.916} C_VEL
LIN {X 0,Y 372.399,Z 532.943,A -85,B 0,C 180,E1 -12870.097,E2 -12870.097} C_VEL
LIN {X 0,Y 373.249,Z 521.119,A -85,B 0,C 180,E1 -12871.079,E2 -12871.079} C_VEL
LIN {X 0,Y 373.893,Z 509.356,A -85,B 0,C 180,E1 -12871.818,E2 -12871.818} C_VEL
LIN {X 0,Y 374.414,Z 496.708,A -85,B 0,C 180,E1 -12872.387,E2 -12872.387} C_VEL
LIN {X 0,Y 374.696,Z 483.838,A -85,B 0,C 180,E1 -12872.755,E2 -12872.755} C_VEL
LIN {X 0,Y 375.857,Z 404.98,A -85,B 0,C 180,E1 -12874.266,E2 -12874.266} C_VEL
LIN {X 0,Y 373.536,Z 393.273,A -85,B 0,C 180,E1 -12874.61,E2 -12874.61} C_VEL
LIN {X 0,Y 371.876,Z 389.685,A -85,B 0,C 180,E1 -12874.779,E2 -12874.779} C_VEL
LIN {X 0,Y 368.55,Z 385.817,A -85,B 0,C 180,E1 -12875.121,E2 -12875.121} C_VEL
LIN {X 0,Y 365.158,Z 382.662,A -85,B 0,C 180,E1 -12875.6,E2 -12875.6} C_VEL
LIN {X 0,Y 363.263,Z 380.532,A -85,B 0,C 180,E1 -12876.066,E2 -12876.066} C_VEL
LIN {X 0,Y 362.665,Z 379.195,A -85,B 0,C 180,E1 -12876.426,E2 -12876.426} C_VEL
LIN {X 0,Y 362.135,Z 376.378,A -85,B 0,C 180,E1 -12877.317,E2 -12877.317} C_VEL
LIN {X 0,Y 361.977,Z 376.396,A -85,B 0,C 180,E1 -12881.195,E2 -12881.195} C_VEL
LIN {X 0,Y 361.966,Z 376.394,A -85,B 0,C 180,E1 -12884.62,E2 -12884.62} C_VEL
LIN {X 0,Y 361.96,Z 376.394,A -85,B 0,C 180,E1 -12888.099,E2 -12888.099} C_VEL
LIN {X 0,Y 361.897,Z 376.405,A -85,B 0,C 180,E1 -12891.652,E2 -12891.652} C_VEL
LIN {X 0,Y 361.931,Z 376.404,A -85,B 0,C 180,E1 -12895.289,E2 -12895.289} C_VEL
LIN {X 0,Y 361.921,Z 376.4,A -85,B 0,C 180,E1 -12897.777,E2 -12897.777} C_VEL
LIN {X 0,Y 361.849,Z 376.413,A -85,B 0,C 180,E1 -12901.284,E2 -12901.284} C_VEL
LIN {X 0,Y 361.856,Z 376.407,A -85,B 0,C 180,E1 -12904.279,E2 -12904.279} C_VEL
LIN {X 0,Y 361.866,Z 376.411,A -85,B 0,C 180,E1 -12907.222,E2 -12907.222} C_VEL
LIN {X 0,Y 361.836,Z 376.413,A -85,B 0,C 180,E1 -12910.755,E2 -12910.755} C_VEL
LIN {X 0,Y 361.833,Z 376.411,A -85,B 0,C 180,E1 -12914.365,E2 -12914.365} C_VEL
LIN {X 0,Y 361.834,Z 376.411,A -85,B 0,C 180,E1 -12917.567,E2 -12917.567} C_VEL
LIN {X 0,Y 361.869,Z 376.412,A -85,B 0,C 180,E1 -12920.972,E2 -12920.972} C_VEL
LIN {X 0,Y 361.871,Z 376.409,A -85,B 0,C 180,E1 -12924.654,E2 -12924.654} C_VEL
LIN {X 0,Y 361.833,Z 376.411,A -85,B 0,C 180,E1 -12928.37,E2 -12928.37} C_VEL
LIN {X 0,Y 361.903,Z 376.402,A -85,B 0,C 180,E1 -12932.22,E2 -12932.22} C_VEL
LIN {X 0,Y 361.923,Z 376.404,A -85,B 0,C 180,E1 -12934.709,E2 -12934.709} C_VEL
LIN {X 0,Y 361.886,Z 376.406,A -85,B 0,C 180,E1 -12938.346,E2 -12938.346} C_VEL
LIN {X 0,Y 361.961,Z 376.395,A -85,B 0,C 180,E1 -12942.061,E2 -12942.061} C_VEL
LIN {X 0,Y 361.991,Z 376.391,A -85,B 0,C 180,E1 -12946.101,E2 -12946.101} C_VEL
LIN {X 0,Y 362.024,Z 376.387,A -85,B 0,C 180,E1 -12949.937,E2 -12949.937} C_VEL
LIN {X 0,Y 362.156,Z 376.37,A -85,B 0,C 180,E1 -12953.313,E2 -12953.313} C_VEL
LIN {X 0,Y 362.275,Z 376.355,A -85,B 0,C 180,E1 -12957.776,E2 -12957.776} C_VEL
LIN {X 0,Y 362.419,Z 376.338,A -85,B 0,C 180,E1 -12960,E2 -12960} C_VEL
LIN {X 0,Y 362.275,Z 376.358,A -85,B 0,C 180,E1 -12962.223,E2 -12962.223} C_VEL
LIN {X 0,Y 362.154,Z 376.374,A -85,B 0,C 180,E1 -12966.686,E2 -12966.686} C_VEL
LIN {X 0,Y 362.023,Z 376.389,A -85,B 0,C 180,E1 -12970.062,E2 -12970.062} C_VEL
LIN {X 0,Y 361.99,Z 376.392,A -85,B 0,C 180,E1 -12973.899,E2 -12973.899} C_VEL
LIN {X 0,Y 361.96,Z 376.397,A -85,B 0,C 180,E1 -12977.939,E2 -12977.939} C_VEL
LIN {X 0,Y 361.885,Z 376.404,A -85,B 0,C 180,E1 -12981.653,E2 -12981.653} C_VEL
LIN {X 0,Y 361.921,Z 376.399,A -85,B 0,C 180,E1 -12985.29,E2 -12985.29} C_VEL
LIN {X 0,Y 361.916,Z 376.402,A -85,B 0,C 180,E1 -12987.778,E2 -12987.778} C_VEL
LIN {X 0,Y 361.841,Z 376.409,A -85,B 0,C 180,E1 -12991.286,E2 -12991.286} C_VEL
LIN {X 0,Y 361.849,Z 376.413,A -85,B 0,C 180,E1 -12994.281,E2 -12994.281} C_VEL
LIN {X 0,Y 361.861,Z 376.407,A -85,B 0,C 180,E1 -12997.224,E2 -12997.224} C_VEL
LIN {X 0,Y 361.902,Z 376.402,A -85,B 0,C 180,E1 -13000.769,E2 -13000.769} C_VEL
LIN {X 0,Y 361.907,Z 376.404,A -85,B 0,C 180,E1 -13004.354,E2 -13004.354} C_VEL
LIN {X 0,Y 361.854,Z 376.409,A -85,B 0,C 180,E1 -13007.565,E2 -13007.565} C_VEL
LIN {X 0,Y 361.872,Z 376.405,A -85,B 0,C 180,E1 -13010.973,E2 -13010.973} C_VEL
LIN {X 0,Y 361.873,Z 376.405,A -85,B 0,C 180,E1 -13014.656,E2 -13014.656} C_VEL
LIN {X 0,Y 361.858,Z 376.408,A -85,B 0,C 180,E1 -13018.373,E2 -13018.373} C_VEL
LIN {X 0,Y 361.925,Z 376.509,A -85,B 0,C 180,E1 -13020.045,E2 -13020.045} C_VEL
LIN {X 0,Y 364.121,Z 386.957,A -85,B 0,C 180,E1 -13022.606,E2 -13022.606} C_VEL
LIN {X 0,Y 365.509,Z 395.643,A -85,B 0,C 180,E1 -13024.651,E2 -13024.651} C_VEL
LIN {X 0,Y 363.945,Z 413.129,A -85,B 0,C 180,E1 -13028.476,E2 -13028.476} C_VEL
